//     PlcTask Inputs/GVL_iXlinker.EtherCAT_Master_EPPxxxx.Beckhoff_EPP2xxx.Beckhoff_EPP2xxxEK1122.A_0016_EPP2304_0061_0018.Channel_2.Input <-> Channel 2/Input
//     PlcTask Outputs/GVL_iXlinker.EtherCAT_Master_EPPxxxx.Beckhoff_EPP2xxx.Beckhoff_EPP2xxxEK1122.A_0016_EPP2304_0061_0018.Channel_3.Output <-> Channel 3/Output
//     PlcTask Outputs/GVL_iXlinker.EtherCAT_Master_EPPxxxx.Beckhoff_EPP2xxx.Beckhoff_EPP2xxxEK1122.A_0016_EPP2304_0061_0018.Channel_4.Output <-> Channel 4/Output
//     PlcTask Inputs/GVL_iXlinker.EtherCAT_Master_EPPxxxx.Beckhoff_EPP2xxx.Beckhoff_EPP2xxxEK1122.A_0016_EPP2304_0061_0018.WcState.WcState <-> WcState/WcState
//     PlcTask Inputs/GVL_iXlinker.EtherCAT_Master_EPPxxxx.Beckhoff_EPP2xxx.Beckhoff_EPP2xxxEK1122.A_0016_EPP2304_0061_0018.WcState.InputToggle <-> WcState/InputToggle
//     PlcTask Inputs/GVL_iXlinker.EtherCAT_Master_EPPxxxx.Beckhoff_EPP2xxx.Beckhoff_EPP2xxxEK1122.A_0016_EPP2304_0061_0018.InfoData.State <-> InfoData/State
//   PLC/PLC Instance <-> EtherCAT Master EPPxxxx/Beckhoff EPP2xxx/Beckhoff EPP2xxxEK1122/A_0017(EPP2308-0001-0016)
//     PlcTask Inputs/GVL_iXlinker.EtherCAT_Master_EPPxxxx.Beckhoff_EPP2xxx.Beckhoff_EPP2xxxEK1122.A_0017_EPP2308_0001_0016.Channel_1.Input <-> Channel 1/Input
//     PlcTask Inputs/GVL_iXlinker.EtherCAT_Master_EPPxxxx.Beckhoff_EPP2xxx.Beckhoff_EPP2xxxEK1122.A_0017_EPP2308_0001_0016.Channel_2.Input <-> Channel 2/Input
//     PlcTask Inputs/GVL_iXlinker.EtherCAT_Master_EPPxxxx.Beckhoff_EPP2xxx.Beckhoff_EPP2xxxEK1122.A_0017_EPP2308_0001_0016.Channel_3.Input <-> Channel 3/Input
//     PlcTask Inputs/GVL_iXlinker.EtherCAT_Master_EPPxxxx.Beckhoff_EPP2xxx.Beckhoff_EPP2xxxEK1122.A_0017_EPP2308_0001_0016.Channel_4.Input <-> Channel 4/Input
//     PlcTask Outputs/GVL_iXlinker.EtherCAT_Master_EPPxxxx.Beckhoff_EPP2xxx.Beckhoff_EPP2xxxEK1122.A_0017_EPP2308_0001_0016.Channel_5.Output <-> Channel 5/Output
//     PlcTask Outputs/GVL_iXlinker.EtherCAT_Master_EPPxxxx.Beckhoff_EPP2xxx.Beckhoff_EPP2xxxEK1122.A_0017_EPP2308_0001_0016.Channel_6.Output <-> Channel 6/Output
//     PlcTask Outputs/GVL_iXlinker.EtherCAT_Master_EPPxxxx.Beckhoff_EPP2xxx.Beckhoff_EPP2xxxEK1122.A_0017_EPP2308_0001_0016.Channel_7.Output <-> Channel 7/Output
//     PlcTask Outputs/GVL_iXlinker.EtherCAT_Master_EPPxxxx.Beckhoff_EPP2xxx.Beckhoff_EPP2xxxEK1122.A_0017_EPP2308_0001_0016.Channel_8.Output <-> Channel 8/Output
//     PlcTask Inputs/GVL_iXlinker.EtherCAT_Master_EPPxxxx.Beckhoff_EPP2xxx.Beckhoff_EPP2xxxEK1122.A_0017_EPP2308_0001_0016.WcState.WcState <-> WcState/WcState
//     PlcTask Inputs/GVL_iXlinker.EtherCAT_Master_EPPxxxx.Beckhoff_EPP2xxx.Beckhoff_EPP2xxxEK1122.A_0017_EPP2308_0001_0016.WcState.InputToggle <-> WcState/InputToggle
//     PlcTask Inputs/GVL_iXlinker.EtherCAT_Master_EPPxxxx.Beckhoff_EPP2xxx.Beckhoff_EPP2xxxEK1122.A_0017_EPP2308_0001_0016.InfoData.State <-> InfoData/State
//   PLC/PLC Instance <-> EtherCAT Master EPPxxxx/Beckhoff EPP2xxx/Beckhoff EPP2xxxEK1122/A_0018(EPP2308-0001-0017)
//     PlcTask Inputs/GVL_iXlinker.EtherCAT_Master_EPPxxxx.Beckhoff_EPP2xxx.Beckhoff_EPP2xxxEK1122.A_0018_EPP2308_0001_0017.Channel_1.Input <-> Channel 1/Input
//     PlcTask Inputs/GVL_iXlinker.EtherCAT_Master_EPPxxxx.Beckhoff_EPP2xxx.Beckhoff_EPP2xxxEK1122.A_0018_EPP2308_0001_0017.Channel_2.Input <-> Channel 2/Input
//     PlcTask Inputs/GVL_iXlinker.EtherCAT_Master_EPPxxxx.Beckhoff_EPP2xxx.Beckhoff_EPP2xxxEK1122.A_0018_EPP2308_0001_0017.Channel_3.Input <-> Channel 3/Input
//     PlcTask Inputs/GVL_iXlinker.EtherCAT_Master_EPPxxxx.Beckhoff_EPP2xxx.Beckhoff_EPP2xxxEK1122.A_0018_EPP2308_0001_0017.Channel_4.Input <-> Channel 4/Input
//     PlcTask Outputs/GVL_iXlinker.EtherCAT_Master_EPPxxxx.Beckhoff_EPP2xxx.Beckhoff_EPP2xxxEK1122.A_0018_EPP2308_0001_0017.Channel_5.Output <-> Channel 5/Output
//     PlcTask Outputs/GVL_iXlinker.EtherCAT_Master_EPPxxxx.Beckhoff_EPP2xxx.Beckhoff_EPP2xxxEK1122.A_0018_EPP2308_0001_0017.Channel_6.Output <-> Channel 6/Output
//     PlcTask Outputs/GVL_iXlinker.EtherCAT_Master_EPPxxxx.Beckhoff_EPP2xxx.Beckhoff_EPP2xxxEK1122.A_0018_EPP2308_0001_0017.Channel_7.Output <-> Channel 7/Output
//     PlcTask Outputs/GVL_iXlinker.EtherCAT_Master_EPPxxxx.Beckhoff_EPP2xxx.Beckhoff_EPP2xxxEK1122.A_0018_EPP2308_0001_0017.Channel_8.Output <-> Channel 8/Output
//     PlcTask Inputs/GVL_iXlinker.EtherCAT_Master_EPPxxxx.Beckhoff_EPP2xxx.Beckhoff_EPP2xxxEK1122.A_0018_EPP2308_0001_0017.WcState.WcState <-> WcState/WcState
//     PlcTask Inputs/GVL_iXlinker.EtherCAT_Master_EPPxxxx.Beckhoff_EPP2xxx.Beckhoff_EPP2xxxEK1122.A_0018_EPP2308_0001_0017.WcState.InputToggle <-> WcState/InputToggle
//     PlcTask Inputs/GVL_iXlinker.EtherCAT_Master_EPPxxxx.Beckhoff_EPP2xxx.Beckhoff_EPP2xxxEK1122.A_0018_EPP2308_0001_0017.InfoData.State <-> InfoData/State
//   PLC/PLC Instance <-> EtherCAT Master EPPxxxx/Beckhoff EPP2xxx/Beckhoff EPP2xxxEK1122/A_0019(EPP2308-0001-0018)
//     PlcTask Inputs/GVL_iXlinker.EtherCAT_Master_EPPxxxx.Beckhoff_EPP2xxx.Beckhoff_EPP2xxxEK1122.A_0019_EPP2308_0001_0018.Channel_1.Input <-> Channel 1/Input
//     PlcTask Inputs/GVL_iXlinker.EtherCAT_Master_EPPxxxx.Beckhoff_EPP2xxx.Beckhoff_EPP2xxxEK1122.A_0019_EPP2308_0001_0018.Channel_2.Input <-> Channel 2/Input
//     PlcTask Inputs/GVL_iXlinker.EtherCAT_Master_EPPxxxx.Beckhoff_EPP2xxx.Beckhoff_EPP2xxxEK1122.A_0019_EPP2308_0001_0018.Channel_3.Input <-> Channel 3/Input
//     PlcTask Inputs/GVL_iXlinker.EtherCAT_Master_EPPxxxx.Beckhoff_EPP2xxx.Beckhoff_EPP2xxxEK1122.A_0019_EPP2308_0001_0018.Channel_4.Input <-> Channel 4/Input
//     PlcTask Outputs/GVL_iXlinker.EtherCAT_Master_EPPxxxx.Beckhoff_EPP2xxx.Beckhoff_EPP2xxxEK1122.A_0019_EPP2308_0001_0018.Channel_5.Output <-> Channel 5/Output
//     PlcTask Outputs/GVL_iXlinker.EtherCAT_Master_EPPxxxx.Beckhoff_EPP2xxx.Beckhoff_EPP2xxxEK1122.A_0019_EPP2308_0001_0018.Channel_6.Output <-> Channel 6/Output
//     PlcTask Outputs/GVL_iXlinker.EtherCAT_Master_EPPxxxx.Beckhoff_EPP2xxx.Beckhoff_EPP2xxxEK1122.A_0019_EPP2308_0001_0018.Channel_7.Output <-> Channel 7/Output
//     PlcTask Outputs/GVL_iXlinker.EtherCAT_Master_EPPxxxx.Beckhoff_EPP2xxx.Beckhoff_EPP2xxxEK1122.A_0019_EPP2308_0001_0018.Channel_8.Output <-> Channel 8/Output
//     PlcTask Inputs/GVL_iXlinker.EtherCAT_Master_EPPxxxx.Beckhoff_EPP2xxx.Beckhoff_EPP2xxxEK1122.A_0019_EPP2308_0001_0018.WcState.WcState <-> WcState/WcState
//     PlcTask Inputs/GVL_iXlinker.EtherCAT_Master_EPPxxxx.Beckhoff_EPP2xxx.Beckhoff_EPP2xxxEK1122.A_0019_EPP2308_0001_0018.WcState.InputToggle <-> WcState/InputToggle
//     PlcTask Inputs/GVL_iXlinker.EtherCAT_Master_EPPxxxx.Beckhoff_EPP2xxx.Beckhoff_EPP2xxxEK1122.A_0019_EPP2308_0001_0018.InfoData.State <-> InfoData/State
//   PLC/PLC Instance <-> EtherCAT Master EPPxxxx/Beckhoff EPP2xxx/Beckhoff EPP2xxxEK1122/A_0020(EPP2308-0002-0016)
//     PlcTask Inputs/GVL_iXlinker.EtherCAT_Master_EPPxxxx.Beckhoff_EPP2xxx.Beckhoff_EPP2xxxEK1122.A_0020_EPP2308_0002_0016.Channel_1.Input <-> Channel 1/Input
//     PlcTask Inputs/GVL_iXlinker.EtherCAT_Master_EPPxxxx.Beckhoff_EPP2xxx.Beckhoff_EPP2xxxEK1122.A_0020_EPP2308_0002_0016.Channel_2.Input <-> Channel 2/Input
//     PlcTask Inputs/GVL_iXlinker.EtherCAT_Master_EPPxxxx.Beckhoff_EPP2xxx.Beckhoff_EPP2xxxEK1122.A_0020_EPP2308_0002_0016.Channel_3.Input <-> Channel 3/Input
//     PlcTask Inputs/GVL_iXlinker.EtherCAT_Master_EPPxxxx.Beckhoff_EPP2xxx.Beckhoff_EPP2xxxEK1122.A_0020_EPP2308_0002_0016.Channel_4.Input <-> Channel 4/Input
//     PlcTask Outputs/GVL_iXlinker.EtherCAT_Master_EPPxxxx.Beckhoff_EPP2xxx.Beckhoff_EPP2xxxEK1122.A_0020_EPP2308_0002_0016.Channel_5.Output <-> Channel 5/Output
//     PlcTask Outputs/GVL_iXlinker.EtherCAT_Master_EPPxxxx.Beckhoff_EPP2xxx.Beckhoff_EPP2xxxEK1122.A_0020_EPP2308_0002_0016.Channel_6.Output <-> Channel 6/Output
//     PlcTask Outputs/GVL_iXlinker.EtherCAT_Master_EPPxxxx.Beckhoff_EPP2xxx.Beckhoff_EPP2xxxEK1122.A_0020_EPP2308_0002_0016.Channel_7.Output <-> Channel 7/Output
//     PlcTask Outputs/GVL_iXlinker.EtherCAT_Master_EPPxxxx.Beckhoff_EPP2xxx.Beckhoff_EPP2xxxEK1122.A_0020_EPP2308_0002_0016.Channel_8.Output <-> Channel 8/Output
//     PlcTask Inputs/GVL_iXlinker.EtherCAT_Master_EPPxxxx.Beckhoff_EPP2xxx.Beckhoff_EPP2xxxEK1122.A_0020_EPP2308_0002_0016.WcState.WcState <-> WcState/WcState
//     PlcTask Inputs/GVL_iXlinker.EtherCAT_Master_EPPxxxx.Beckhoff_EPP2xxx.Beckhoff_EPP2xxxEK1122.A_0020_EPP2308_0002_0016.WcState.InputToggle <-> WcState/InputToggle
//     PlcTask Inputs/GVL_iXlinker.EtherCAT_Master_EPPxxxx.Beckhoff_EPP2xxx.Beckhoff_EPP2xxxEK1122.A_0020_EPP2308_0002_0016.InfoData.State <-> InfoData/State
//   PLC/PLC Instance <-> EtherCAT Master EPPxxxx/Beckhoff EPP2xxx/Beckhoff EPP2xxxEK1122/A_0021(EPP2308-0002-0017)
//     PlcTask Inputs/GVL_iXlinker.EtherCAT_Master_EPPxxxx.Beckhoff_EPP2xxx.Beckhoff_EPP2xxxEK1122.A_0021_EPP2308_0002_0017.Channel_1.Input <-> Channel 1/Input
//     PlcTask Inputs/GVL_iXlinker.EtherCAT_Master_EPPxxxx.Beckhoff_EPP2xxx.Beckhoff_EPP2xxxEK1122.A_0021_EPP2308_0002_0017.Channel_2.Input <-> Channel 2/Input
//     PlcTask Inputs/GVL_iXlinker.EtherCAT_Master_EPPxxxx.Beckhoff_EPP2xxx.Beckhoff_EPP2xxxEK1122.A_0021_EPP2308_0002_0017.Channel_3.Input <-> Channel 3/Input
//     PlcTask Inputs/GVL_iXlinker.EtherCAT_Master_EPPxxxx.Beckhoff_EPP2xxx.Beckhoff_EPP2xxxEK1122.A_0021_EPP2308_0002_0017.Channel_4.Input <-> Channel 4/Input
//     PlcTask Outputs/GVL_iXlinker.EtherCAT_Master_EPPxxxx.Beckhoff_EPP2xxx.Beckhoff_EPP2xxxEK1122.A_0021_EPP2308_0002_0017.Channel_5.Output <-> Channel 5/Output
//     PlcTask Outputs/GVL_iXlinker.EtherCAT_Master_EPPxxxx.Beckhoff_EPP2xxx.Beckhoff_EPP2xxxEK1122.A_0021_EPP2308_0002_0017.Channel_6.Output <-> Channel 6/Output
//     PlcTask Outputs/GVL_iXlinker.EtherCAT_Master_EPPxxxx.Beckhoff_EPP2xxx.Beckhoff_EPP2xxxEK1122.A_0021_EPP2308_0002_0017.Channel_7.Output <-> Channel 7/Output
//     PlcTask Outputs/GVL_iXlinker.EtherCAT_Master_EPPxxxx.Beckhoff_EPP2xxx.Beckhoff_EPP2xxxEK1122.A_0021_EPP2308_0002_0017.Channel_8.Output <-> Channel 8/Output
//     PlcTask Inputs/GVL_iXlinker.EtherCAT_Master_EPPxxxx.Beckhoff_EPP2xxx.Beckhoff_EPP2xxxEK1122.A_0021_EPP2308_0002_0017.WcState.WcState <-> WcState/WcState
//     PlcTask Inputs/GVL_iXlinker.EtherCAT_Master_EPPxxxx.Beckhoff_EPP2xxx.Beckhoff_EPP2xxxEK1122.A_0021_EPP2308_0002_0017.WcState.InputToggle <-> WcState/InputToggle
//     PlcTask Inputs/GVL_iXlinker.EtherCAT_Master_EPPxxxx.Beckhoff_EPP2xxx.Beckhoff_EPP2xxxEK1122.A_0021_EPP2308_0002_0017.InfoData.State <-> InfoData/State
//   PLC/PLC Instance <-> EtherCAT Master EPPxxxx/Beckhoff EPP2xxx/Beckhoff EPP2xxxEK1122/A_0022(EPP2308-0002-0018)
//     PlcTask Inputs/GVL_iXlinker.EtherCAT_Master_EPPxxxx.Beckhoff_EPP2xxx.Beckhoff_EPP2xxxEK1122.A_0022_EPP2308_0002_0018.Channel_1.Input <-> Channel 1/Input
//     PlcTask Inputs/GVL_iXlinker.EtherCAT_Master_EPPxxxx.Beckhoff_EPP2xxx.Beckhoff_EPP2xxxEK1122.A_0022_EPP2308_0002_0018.Channel_2.Input <-> Channel 2/Input
//     PlcTask Inputs/GVL_iXlinker.EtherCAT_Master_EPPxxxx.Beckhoff_EPP2xxx.Beckhoff_EPP2xxxEK1122.A_0022_EPP2308_0002_0018.Channel_3.Input <-> Channel 3/Input
//     PlcTask Inputs/GVL_iXlinker.EtherCAT_Master_EPPxxxx.Beckhoff_EPP2xxx.Beckhoff_EPP2xxxEK1122.A_0022_EPP2308_0002_0018.Channel_4.Input <-> Channel 4/Input
//     PlcTask Outputs/GVL_iXlinker.EtherCAT_Master_EPPxxxx.Beckhoff_EPP2xxx.Beckhoff_EPP2xxxEK1122.A_0022_EPP2308_0002_0018.Channel_5.Output <-> Channel 5/Output
//     PlcTask Outputs/GVL_iXlinker.EtherCAT_Master_EPPxxxx.Beckhoff_EPP2xxx.Beckhoff_EPP2xxxEK1122.A_0022_EPP2308_0002_0018.Channel_6.Output <-> Channel 6/Output
//     PlcTask Outputs/GVL_iXlinker.EtherCAT_Master_EPPxxxx.Beckhoff_EPP2xxx.Beckhoff_EPP2xxxEK1122.A_0022_EPP2308_0002_0018.Channel_7.Output <-> Channel 7/Output
//     PlcTask Outputs/GVL_iXlinker.EtherCAT_Master_EPPxxxx.Beckhoff_EPP2xxx.Beckhoff_EPP2xxxEK1122.A_0022_EPP2308_0002_0018.Channel_8.Output <-> Channel 8/Output
//     PlcTask Inputs/GVL_iXlinker.EtherCAT_Master_EPPxxxx.Beckhoff_EPP2xxx.Beckhoff_EPP2xxxEK1122.A_0022_EPP2308_0002_0018.WcState.WcState <-> WcState/WcState
//     PlcTask Inputs/GVL_iXlinker.EtherCAT_Master_EPPxxxx.Beckhoff_EPP2xxx.Beckhoff_EPP2xxxEK1122.A_0022_EPP2308_0002_0018.WcState.InputToggle <-> WcState/InputToggle
//     PlcTask Inputs/GVL_iXlinker.EtherCAT_Master_EPPxxxx.Beckhoff_EPP2xxx.Beckhoff_EPP2xxxEK1122.A_0022_EPP2308_0002_0018.InfoData.State <-> InfoData/State
//   PLC/PLC Instance <-> EtherCAT Master EPPxxxx/Beckhoff EPP2xxx/Beckhoff EPP2xxxEK1122/A_0023(EPP2316-0003-0016)
//     PlcTask Inputs/GVL_iXlinker.EtherCAT_Master_EPPxxxx.Beckhoff_EPP2xxx.Beckhoff_EPP2xxxEK1122.A_0023_EPP2316_0003_0016.DIG_Inputs.Input[0] <-> DIG Inputs/Input 1
//     PlcTask Inputs/GVL_iXlinker.EtherCAT_Master_EPPxxxx.Beckhoff_EPP2xxx.Beckhoff_EPP2xxxEK1122.A_0023_EPP2316_0003_0016.DIG_Inputs.Input[1] <-> DIG Inputs/Input 2
//     PlcTask Inputs/GVL_iXlinker.EtherCAT_Master_EPPxxxx.Beckhoff_EPP2xxx.Beckhoff_EPP2xxxEK1122.A_0023_EPP2316_0003_0016.DIG_Inputs.Input[2] <-> DIG Inputs/Input 3
//     PlcTask Inputs/GVL_iXlinker.EtherCAT_Master_EPPxxxx.Beckhoff_EPP2xxx.Beckhoff_EPP2xxxEK1122.A_0023_EPP2316_0003_0016.DIG_Inputs.Input[3] <-> DIG Inputs/Input 4
//     PlcTask Inputs/GVL_iXlinker.EtherCAT_Master_EPPxxxx.Beckhoff_EPP2xxx.Beckhoff_EPP2xxxEK1122.A_0023_EPP2316_0003_0016.DIG_Inputs.Input[4] <-> DIG Inputs/Input 5
//     PlcTask Inputs/GVL_iXlinker.EtherCAT_Master_EPPxxxx.Beckhoff_EPP2xxx.Beckhoff_EPP2xxxEK1122.A_0023_EPP2316_0003_0016.DIG_Inputs.Input[5] <-> DIG Inputs/Input 6
//     PlcTask Inputs/GVL_iXlinker.EtherCAT_Master_EPPxxxx.Beckhoff_EPP2xxx.Beckhoff_EPP2xxxEK1122.A_0023_EPP2316_0003_0016.DIG_Inputs.Input[6] <-> DIG Inputs/Input 7
//     PlcTask Inputs/GVL_iXlinker.EtherCAT_Master_EPPxxxx.Beckhoff_EPP2xxx.Beckhoff_EPP2xxxEK1122.A_0023_EPP2316_0003_0016.DIG_Inputs.Input[7] <-> DIG Inputs/Input 8
//     PlcTask Inputs/GVL_iXlinker.EtherCAT_Master_EPPxxxx.Beckhoff_EPP2xxx.Beckhoff_EPP2xxxEK1122.A_0023_EPP2316_0003_0016.DIG_Inputs.Sync_Error <-> DIG Inputs/Sync Error
//     PlcTask Inputs/GVL_iXlinker.EtherCAT_Master_EPPxxxx.Beckhoff_EPP2xxx.Beckhoff_EPP2xxxEK1122.A_0023_EPP2316_0003_0016.DIG_Diag_Inputs.Diag_Input[0] <-> DIG Diag Inputs/Diag Input 1
//     PlcTask Inputs/GVL_iXlinker.EtherCAT_Master_EPPxxxx.Beckhoff_EPP2xxx.Beckhoff_EPP2xxxEK1122.A_0023_EPP2316_0003_0016.DIG_Diag_Inputs.Diag_Input[1] <-> DIG Diag Inputs/Diag Input 2
//     PlcTask Inputs/GVL_iXlinker.EtherCAT_Master_EPPxxxx.Beckhoff_EPP2xxx.Beckhoff_EPP2xxxEK1122.A_0023_EPP2316_0003_0016.DIG_Diag_Inputs.Diag_Input[2] <-> DIG Diag Inputs/Diag Input 3
//     PlcTask Inputs/GVL_iXlinker.EtherCAT_Master_EPPxxxx.Beckhoff_EPP2xxx.Beckhoff_EPP2xxxEK1122.A_0023_EPP2316_0003_0016.DIG_Diag_Inputs.Diag_Input[3] <-> DIG Diag Inputs/Diag Input 4
//     PlcTask Inputs/GVL_iXlinker.EtherCAT_Master_EPPxxxx.Beckhoff_EPP2xxx.Beckhoff_EPP2xxxEK1122.A_0023_EPP2316_0003_0016.DIG_Diag_Inputs.Diag_Input[4] <-> DIG Diag Inputs/Diag Input 5
//     PlcTask Inputs/GVL_iXlinker.EtherCAT_Master_EPPxxxx.Beckhoff_EPP2xxx.Beckhoff_EPP2xxxEK1122.A_0023_EPP2316_0003_0016.DIG_Diag_Inputs.Diag_Input[5] <-> DIG Diag Inputs/Diag Input 6
//     PlcTask Inputs/GVL_iXlinker.EtherCAT_Master_EPPxxxx.Beckhoff_EPP2xxx.Beckhoff_EPP2xxxEK1122.A_0023_EPP2316_0003_0016.DIG_Diag_Inputs.Diag_Input[6] <-> DIG Diag Inputs/Diag Input 7
//     PlcTask Inputs/GVL_iXlinker.EtherCAT_Master_EPPxxxx.Beckhoff_EPP2xxx.Beckhoff_EPP2xxxEK1122.A_0023_EPP2316_0003_0016.DIG_Diag_Inputs.Diag_Input[7] <-> DIG Diag Inputs/Diag Input 8
//     PlcTask Inputs/GVL_iXlinker.EtherCAT_Master_EPPxxxx.Beckhoff_EPP2xxx.Beckhoff_EPP2xxxEK1122.A_0023_EPP2316_0003_0016.DIG_Inputs_Device.Safe_state_active <-> DIG Inputs Device/Safe state active
//     PlcTask Inputs/GVL_iXlinker.EtherCAT_Master_EPPxxxx.Beckhoff_EPP2xxx.Beckhoff_EPP2xxxEK1122.A_0023_EPP2316_0003_0016.DIG_Inputs_Device.Error_channel[0] <-> DIG Inputs Device/Error channel 1
//     PlcTask Inputs/GVL_iXlinker.EtherCAT_Master_EPPxxxx.Beckhoff_EPP2xxx.Beckhoff_EPP2xxxEK1122.A_0023_EPP2316_0003_0016.DIG_Inputs_Device.Error_channel[1] <-> DIG Inputs Device/Error channel 2
//     PlcTask Inputs/GVL_iXlinker.EtherCAT_Master_EPPxxxx.Beckhoff_EPP2xxx.Beckhoff_EPP2xxxEK1122.A_0023_EPP2316_0003_0016.DIG_Inputs_Device.Sync_error <-> DIG Inputs Device/Sync error
//     PlcTask Inputs/GVL_iXlinker.EtherCAT_Master_EPPxxxx.Beckhoff_EPP2xxx.Beckhoff_EPP2xxxEK1122.A_0023_EPP2316_0003_0016.DIG_Inputs_Device.TxPDO_Toggle <-> DIG Inputs Device/TxPDO Toggle
//     PlcTask Outputs/GVL_iXlinker.EtherCAT_Master_EPPxxxx.Beckhoff_EPP2xxx.Beckhoff_EPP2xxxEK1122.A_0023_EPP2316_0003_0016.DIG_Outputs.Output[0] <-> DIG Outputs/Output 1
//     PlcTask Outputs/GVL_iXlinker.EtherCAT_Master_EPPxxxx.Beckhoff_EPP2xxx.Beckhoff_EPP2xxxEK1122.A_0023_EPP2316_0003_0016.DIG_Outputs.Output[1] <-> DIG Outputs/Output 2
//     PlcTask Outputs/GVL_iXlinker.EtherCAT_Master_EPPxxxx.Beckhoff_EPP2xxx.Beckhoff_EPP2xxxEK1122.A_0023_EPP2316_0003_0016.DIG_Outputs.Output[2] <-> DIG Outputs/Output 3
//     PlcTask Outputs/GVL_iXlinker.EtherCAT_Master_EPPxxxx.Beckhoff_EPP2xxx.Beckhoff_EPP2xxxEK1122.A_0023_EPP2316_0003_0016.DIG_Outputs.Output[3] <-> DIG Outputs/Output 4
//     PlcTask Outputs/GVL_iXlinker.EtherCAT_Master_EPPxxxx.Beckhoff_EPP2xxx.Beckhoff_EPP2xxxEK1122.A_0023_EPP2316_0003_0016.DIG_Outputs.Output[4] <-> DIG Outputs/Output 5
//     PlcTask Outputs/GVL_iXlinker.EtherCAT_Master_EPPxxxx.Beckhoff_EPP2xxx.Beckhoff_EPP2xxxEK1122.A_0023_EPP2316_0003_0016.DIG_Outputs.Output[5] <-> DIG Outputs/Output 6
//     PlcTask Outputs/GVL_iXlinker.EtherCAT_Master_EPPxxxx.Beckhoff_EPP2xxx.Beckhoff_EPP2xxxEK1122.A_0023_EPP2316_0003_0016.DIG_Outputs.Output[6] <-> DIG Outputs/Output 7
//     PlcTask Outputs/GVL_iXlinker.EtherCAT_Master_EPPxxxx.Beckhoff_EPP2xxx.Beckhoff_EPP2xxxEK1122.A_0023_EPP2316_0003_0016.DIG_Outputs.Output[7] <-> DIG Outputs/Output 8
//     PlcTask Outputs/GVL_iXlinker.EtherCAT_Master_EPPxxxx.Beckhoff_EPP2xxx.Beckhoff_EPP2xxxEK1122.A_0023_EPP2316_0003_0016.DIG_Outputs_Device.Set_safe_state <-> DIG Outputs Device/Set safe state
//     PlcTask Outputs/GVL_iXlinker.EtherCAT_Master_EPPxxxx.Beckhoff_EPP2xxx.Beckhoff_EPP2xxxEK1122.A_0023_EPP2316_0003_0016.DIG_Outputs_Device.Reset_outputs <-> DIG Outputs Device/Reset outputs
//     PlcTask Inputs/GVL_iXlinker.EtherCAT_Master_EPPxxxx.Beckhoff_EPP2xxx.Beckhoff_EPP2xxxEK1122.A_0023_EPP2316_0003_0016.WcState.WcState <-> WcState/WcState
//     PlcTask Inputs/GVL_iXlinker.EtherCAT_Master_EPPxxxx.Beckhoff_EPP2xxx.Beckhoff_EPP2xxxEK1122.A_0023_EPP2316_0003_0016.WcState.InputToggle <-> WcState/InputToggle
//     PlcTask Inputs/GVL_iXlinker.EtherCAT_Master_EPPxxxx.Beckhoff_EPP2xxx.Beckhoff_EPP2xxxEK1122.A_0023_EPP2316_0003_0016.InfoData.AdsAddr <-> InfoData/AdsAddr
//     PlcTask Inputs/GVL_iXlinker.EtherCAT_Master_EPPxxxx.Beckhoff_EPP2xxx.Beckhoff_EPP2xxxEK1122.A_0023_EPP2316_0003_0016.InfoData.State <-> InfoData/State
//   PLC/PLC Instance <-> EtherCAT Master EPPxxxx/Beckhoff EPP2xxx/Beckhoff EPP2xxxEK1122/A_0024(EPP2316-0003-0017)
//     PlcTask Inputs/GVL_iXlinker.EtherCAT_Master_EPPxxxx.Beckhoff_EPP2xxx.Beckhoff_EPP2xxxEK1122.A_0024_EPP2316_0003_0017.DIG_Inputs.Input[0] <-> DIG Inputs/Input 1
//     PlcTask Inputs/GVL_iXlinker.EtherCAT_Master_EPPxxxx.Beckhoff_EPP2xxx.Beckhoff_EPP2xxxEK1122.A_0024_EPP2316_0003_0017.DIG_Inputs.Input[1] <-> DIG Inputs/Input 2
//     PlcTask Inputs/GVL_iXlinker.EtherCAT_Master_EPPxxxx.Beckhoff_EPP2xxx.Beckhoff_EPP2xxxEK1122.A_0024_EPP2316_0003_0017.DIG_Inputs.Input[2] <-> DIG Inputs/Input 3
//     PlcTask Inputs/GVL_iXlinker.EtherCAT_Master_EPPxxxx.Beckhoff_EPP2xxx.Beckhoff_EPP2xxxEK1122.A_0024_EPP2316_0003_0017.DIG_Inputs.Input[3] <-> DIG Inputs/Input 4
//     PlcTask Inputs/GVL_iXlinker.EtherCAT_Master_EPPxxxx.Beckhoff_EPP2xxx.Beckhoff_EPP2xxxEK1122.A_0024_EPP2316_0003_0017.DIG_Inputs.Input[4] <-> DIG Inputs/Input 5
//     PlcTask Inputs/GVL_iXlinker.EtherCAT_Master_EPPxxxx.Beckhoff_EPP2xxx.Beckhoff_EPP2xxxEK1122.A_0024_EPP2316_0003_0017.DIG_Inputs.Input[5] <-> DIG Inputs/Input 6
//     PlcTask Inputs/GVL_iXlinker.EtherCAT_Master_EPPxxxx.Beckhoff_EPP2xxx.Beckhoff_EPP2xxxEK1122.A_0024_EPP2316_0003_0017.DIG_Inputs.Input[6] <-> DIG Inputs/Input 7
//     PlcTask Inputs/GVL_iXlinker.EtherCAT_Master_EPPxxxx.Beckhoff_EPP2xxx.Beckhoff_EPP2xxxEK1122.A_0024_EPP2316_0003_0017.DIG_Inputs.Input[7] <-> DIG Inputs/Input 8
//     PlcTask Inputs/GVL_iXlinker.EtherCAT_Master_EPPxxxx.Beckhoff_EPP2xxx.Beckhoff_EPP2xxxEK1122.A_0024_EPP2316_0003_0017.DIG_Inputs.Sync_Error <-> DIG Inputs/Sync Error
//     PlcTask Inputs/GVL_iXlinker.EtherCAT_Master_EPPxxxx.Beckhoff_EPP2xxx.Beckhoff_EPP2xxxEK1122.A_0024_EPP2316_0003_0017.DIG_Diag_Inputs.Diag_Input[0] <-> DIG Diag Inputs/Diag Input 1
//     PlcTask Inputs/GVL_iXlinker.EtherCAT_Master_EPPxxxx.Beckhoff_EPP2xxx.Beckhoff_EPP2xxxEK1122.A_0024_EPP2316_0003_0017.DIG_Diag_Inputs.Diag_Input[1] <-> DIG Diag Inputs/Diag Input 2
//     PlcTask Inputs/GVL_iXlinker.EtherCAT_Master_EPPxxxx.Beckhoff_EPP2xxx.Beckhoff_EPP2xxxEK1122.A_0024_EPP2316_0003_0017.DIG_Diag_Inputs.Diag_Input[2] <-> DIG Diag Inputs/Diag Input 3
//     PlcTask Inputs/GVL_iXlinker.EtherCAT_Master_EPPxxxx.Beckhoff_EPP2xxx.Beckhoff_EPP2xxxEK1122.A_0024_EPP2316_0003_0017.DIG_Diag_Inputs.Diag_Input[3] <-> DIG Diag Inputs/Diag Input 4
//     PlcTask Inputs/GVL_iXlinker.EtherCAT_Master_EPPxxxx.Beckhoff_EPP2xxx.Beckhoff_EPP2xxxEK1122.A_0024_EPP2316_0003_0017.DIG_Diag_Inputs.Diag_Input[4] <-> DIG Diag Inputs/Diag Input 5
//     PlcTask Inputs/GVL_iXlinker.EtherCAT_Master_EPPxxxx.Beckhoff_EPP2xxx.Beckhoff_EPP2xxxEK1122.A_0024_EPP2316_0003_0017.DIG_Diag_Inputs.Diag_Input[5] <-> DIG Diag Inputs/Diag Input 6
//     PlcTask Inputs/GVL_iXlinker.EtherCAT_Master_EPPxxxx.Beckhoff_EPP2xxx.Beckhoff_EPP2xxxEK1122.A_0024_EPP2316_0003_0017.DIG_Diag_Inputs.Diag_Input[6] <-> DIG Diag Inputs/Diag Input 7
//     PlcTask Inputs/GVL_iXlinker.EtherCAT_Master_EPPxxxx.Beckhoff_EPP2xxx.Beckhoff_EPP2xxxEK1122.A_0024_EPP2316_0003_0017.DIG_Diag_Inputs.Diag_Input[7] <-> DIG Diag Inputs/Diag Input 8
//     PlcTask Inputs/GVL_iXlinker.EtherCAT_Master_EPPxxxx.Beckhoff_EPP2xxx.Beckhoff_EPP2xxxEK1122.A_0024_EPP2316_0003_0017.DIG_Inputs_Device.Safe_state_active <-> DIG Inputs Device/Safe state active
//     PlcTask Inputs/GVL_iXlinker.EtherCAT_Master_EPPxxxx.Beckhoff_EPP2xxx.Beckhoff_EPP2xxxEK1122.A_0024_EPP2316_0003_0017.DIG_Inputs_Device.Error_channel[0] <-> DIG Inputs Device/Error channel 1
//     PlcTask Inputs/GVL_iXlinker.EtherCAT_Master_EPPxxxx.Beckhoff_EPP2xxx.Beckhoff_EPP2xxxEK1122.A_0024_EPP2316_0003_0017.DIG_Inputs_Device.Error_channel[1] <-> DIG Inputs Device/Error channel 2
//     PlcTask Inputs/GVL_iXlinker.EtherCAT_Master_EPPxxxx.Beckhoff_EPP2xxx.Beckhoff_EPP2xxxEK1122.A_0024_EPP2316_0003_0017.DIG_Inputs_Device.Sync_error <-> DIG Inputs Device/Sync error
//     PlcTask Inputs/GVL_iXlinker.EtherCAT_Master_EPPxxxx.Beckhoff_EPP2xxx.Beckhoff_EPP2xxxEK1122.A_0024_EPP2316_0003_0017.DIG_Inputs_Device.TxPDO_Toggle <-> DIG Inputs Device/TxPDO Toggle
//     PlcTask Outputs/GVL_iXlinker.EtherCAT_Master_EPPxxxx.Beckhoff_EPP2xxx.Beckhoff_EPP2xxxEK1122.A_0024_EPP2316_0003_0017.DIG_Outputs.Output[0] <-> DIG Outputs/Output 1
//     PlcTask Outputs/GVL_iXlinker.EtherCAT_Master_EPPxxxx.Beckhoff_EPP2xxx.Beckhoff_EPP2xxxEK1122.A_0024_EPP2316_0003_0017.DIG_Outputs.Output[1] <-> DIG Outputs/Output 2
//     PlcTask Outputs/GVL_iXlinker.EtherCAT_Master_EPPxxxx.Beckhoff_EPP2xxx.Beckhoff_EPP2xxxEK1122.A_0024_EPP2316_0003_0017.DIG_Outputs.Output[2] <-> DIG Outputs/Output 3
//     PlcTask Outputs/GVL_iXlinker.EtherCAT_Master_EPPxxxx.Beckhoff_EPP2xxx.Beckhoff_EPP2xxxEK1122.A_0024_EPP2316_0003_0017.DIG_Outputs.Output[3] <-> DIG Outputs/Output 4
//     PlcTask Outputs/GVL_iXlinker.EtherCAT_Master_EPPxxxx.Beckhoff_EPP2xxx.Beckhoff_EPP2xxxEK1122.A_0024_EPP2316_0003_0017.DIG_Outputs.Output[4] <-> DIG Outputs/Output 5
//     PlcTask Outputs/GVL_iXlinker.EtherCAT_Master_EPPxxxx.Beckhoff_EPP2xxx.Beckhoff_EPP2xxxEK1122.A_0024_EPP2316_0003_0017.DIG_Outputs.Output[5] <-> DIG Outputs/Output 6
//     PlcTask Outputs/GVL_iXlinker.EtherCAT_Master_EPPxxxx.Beckhoff_EPP2xxx.Beckhoff_EPP2xxxEK1122.A_0024_EPP2316_0003_0017.DIG_Outputs.Output[6] <-> DIG Outputs/Output 7
//     PlcTask Outputs/GVL_iXlinker.EtherCAT_Master_EPPxxxx.Beckhoff_EPP2xxx.Beckhoff_EPP2xxxEK1122.A_0024_EPP2316_0003_0017.DIG_Outputs.Output[7] <-> DIG Outputs/Output 8
//     PlcTask Outputs/GVL_iXlinker.EtherCAT_Master_EPPxxxx.Beckhoff_EPP2xxx.Beckhoff_EPP2xxxEK1122.A_0024_EPP2316_0003_0017.DIG_Outputs_Device.Set_safe_state <-> DIG Outputs Device/Set safe state
//     PlcTask Outputs/GVL_iXlinker.EtherCAT_Master_EPPxxxx.Beckhoff_EPP2xxx.Beckhoff_EPP2xxxEK1122.A_0024_EPP2316_0003_0017.DIG_Outputs_Device.Reset_outputs <-> DIG Outputs Device/Reset outputs
//     PlcTask Inputs/GVL_iXlinker.EtherCAT_Master_EPPxxxx.Beckhoff_EPP2xxx.Beckhoff_EPP2xxxEK1122.A_0024_EPP2316_0003_0017.WcState.WcState <-> WcState/WcState
//     PlcTask Inputs/GVL_iXlinker.EtherCAT_Master_EPPxxxx.Beckhoff_EPP2xxx.Beckhoff_EPP2xxxEK1122.A_0024_EPP2316_0003_0017.WcState.InputToggle <-> WcState/InputToggle
//     PlcTask Inputs/GVL_iXlinker.EtherCAT_Master_EPPxxxx.Beckhoff_EPP2xxx.Beckhoff_EPP2xxxEK1122.A_0024_EPP2316_0003_0017.InfoData.AdsAddr <-> InfoData/AdsAddr
//     PlcTask Inputs/GVL_iXlinker.EtherCAT_Master_EPPxxxx.Beckhoff_EPP2xxx.Beckhoff_EPP2xxxEK1122.A_0024_EPP2316_0003_0017.InfoData.State <-> InfoData/State
//   PLC/PLC Instance <-> EtherCAT Master EPPxxxx/Beckhoff EPP2xxx/Beckhoff EPP2xxxEK1122/A_0025(EPP2316-0003-0018)
//     PlcTask Inputs/GVL_iXlinker.EtherCAT_Master_EPPxxxx.Beckhoff_EPP2xxx.Beckhoff_EPP2xxxEK1122.A_0025_EPP2316_0003_0018.DIG_Inputs.Input[0] <-> DIG Inputs/Input 1
//     PlcTask Inputs/GVL_iXlinker.EtherCAT_Master_EPPxxxx.Beckhoff_EPP2xxx.Beckhoff_EPP2xxxEK1122.A_0025_EPP2316_0003_0018.DIG_Inputs.Input[1] <-> DIG Inputs/Input 2
//     PlcTask Inputs/GVL_iXlinker.EtherCAT_Master_EPPxxxx.Beckhoff_EPP2xxx.Beckhoff_EPP2xxxEK1122.A_0025_EPP2316_0003_0018.DIG_Inputs.Input[2] <-> DIG Inputs/Input 3
//     PlcTask Inputs/GVL_iXlinker.EtherCAT_Master_EPPxxxx.Beckhoff_EPP2xxx.Beckhoff_EPP2xxxEK1122.A_0025_EPP2316_0003_0018.DIG_Inputs.Input[3] <-> DIG Inputs/Input 4
//     PlcTask Inputs/GVL_iXlinker.EtherCAT_Master_EPPxxxx.Beckhoff_EPP2xxx.Beckhoff_EPP2xxxEK1122.A_0025_EPP2316_0003_0018.DIG_Inputs.Input[4] <-> DIG Inputs/Input 5
//     PlcTask Inputs/GVL_iXlinker.EtherCAT_Master_EPPxxxx.Beckhoff_EPP2xxx.Beckhoff_EPP2xxxEK1122.A_0025_EPP2316_0003_0018.DIG_Inputs.Input[5] <-> DIG Inputs/Input 6
//     PlcTask Inputs/GVL_iXlinker.EtherCAT_Master_EPPxxxx.Beckhoff_EPP2xxx.Beckhoff_EPP2xxxEK1122.A_0025_EPP2316_0003_0018.DIG_Inputs.Input[6] <-> DIG Inputs/Input 7
//     PlcTask Inputs/GVL_iXlinker.EtherCAT_Master_EPPxxxx.Beckhoff_EPP2xxx.Beckhoff_EPP2xxxEK1122.A_0025_EPP2316_0003_0018.DIG_Inputs.Input[7] <-> DIG Inputs/Input 8
//     PlcTask Inputs/GVL_iXlinker.EtherCAT_Master_EPPxxxx.Beckhoff_EPP2xxx.Beckhoff_EPP2xxxEK1122.A_0025_EPP2316_0003_0018.DIG_Inputs.Sync_error <-> DIG Inputs/Sync error
//     PlcTask Inputs/GVL_iXlinker.EtherCAT_Master_EPPxxxx.Beckhoff_EPP2xxx.Beckhoff_EPP2xxxEK1122.A_0025_EPP2316_0003_0018.DIG_Diag_Inputs.Diag_Input[0] <-> DIG Diag Inputs/Diag Input 1
//     PlcTask Inputs/GVL_iXlinker.EtherCAT_Master_EPPxxxx.Beckhoff_EPP2xxx.Beckhoff_EPP2xxxEK1122.A_0025_EPP2316_0003_0018.DIG_Diag_Inputs.Diag_Input[1] <-> DIG Diag Inputs/Diag Input 2
//     PlcTask Inputs/GVL_iXlinker.EtherCAT_Master_EPPxxxx.Beckhoff_EPP2xxx.Beckhoff_EPP2xxxEK1122.A_0025_EPP2316_0003_0018.DIG_Diag_Inputs.Diag_Input[2] <-> DIG Diag Inputs/Diag Input 3
//     PlcTask Inputs/GVL_iXlinker.EtherCAT_Master_EPPxxxx.Beckhoff_EPP2xxx.Beckhoff_EPP2xxxEK1122.A_0025_EPP2316_0003_0018.DIG_Diag_Inputs.Diag_Input[3] <-> DIG Diag Inputs/Diag Input 4
//     PlcTask Inputs/GVL_iXlinker.EtherCAT_Master_EPPxxxx.Beckhoff_EPP2xxx.Beckhoff_EPP2xxxEK1122.A_0025_EPP2316_0003_0018.DIG_Diag_Inputs.Diag_Input[4] <-> DIG Diag Inputs/Diag Input 5
//     PlcTask Inputs/GVL_iXlinker.EtherCAT_Master_EPPxxxx.Beckhoff_EPP2xxx.Beckhoff_EPP2xxxEK1122.A_0025_EPP2316_0003_0018.DIG_Diag_Inputs.Diag_Input[5] <-> DIG Diag Inputs/Diag Input 6
//     PlcTask Inputs/GVL_iXlinker.EtherCAT_Master_EPPxxxx.Beckhoff_EPP2xxx.Beckhoff_EPP2xxxEK1122.A_0025_EPP2316_0003_0018.DIG_Diag_Inputs.Diag_Input[6] <-> DIG Diag Inputs/Diag Input 7
//     PlcTask Inputs/GVL_iXlinker.EtherCAT_Master_EPPxxxx.Beckhoff_EPP2xxx.Beckhoff_EPP2xxxEK1122.A_0025_EPP2316_0003_0018.DIG_Diag_Inputs.Diag_Input[7] <-> DIG Diag Inputs/Diag Input 8
//     PlcTask Inputs/GVL_iXlinker.EtherCAT_Master_EPPxxxx.Beckhoff_EPP2xxx.Beckhoff_EPP2xxxEK1122.A_0025_EPP2316_0003_0018.DIG_Inputs_Device.Safe_state_active <-> DIG Inputs Device/Safe state active
//     PlcTask Inputs/GVL_iXlinker.EtherCAT_Master_EPPxxxx.Beckhoff_EPP2xxx.Beckhoff_EPP2xxxEK1122.A_0025_EPP2316_0003_0018.DIG_Inputs_Device.Error_channel[0] <-> DIG Inputs Device/Error channel 1
//     PlcTask Inputs/GVL_iXlinker.EtherCAT_Master_EPPxxxx.Beckhoff_EPP2xxx.Beckhoff_EPP2xxxEK1122.A_0025_EPP2316_0003_0018.DIG_Inputs_Device.Error_channel[1] <-> DIG Inputs Device/Error channel 2
//     PlcTask Inputs/GVL_iXlinker.EtherCAT_Master_EPPxxxx.Beckhoff_EPP2xxx.Beckhoff_EPP2xxxEK1122.A_0025_EPP2316_0003_0018.DIG_Inputs_Device.Sync_error <-> DIG Inputs Device/Sync error
//     PlcTask Inputs/GVL_iXlinker.EtherCAT_Master_EPPxxxx.Beckhoff_EPP2xxx.Beckhoff_EPP2xxxEK1122.A_0025_EPP2316_0003_0018.DIG_Inputs_Device.TxPDO_Toggle <-> DIG Inputs Device/TxPDO Toggle
//     PlcTask Outputs/GVL_iXlinker.EtherCAT_Master_EPPxxxx.Beckhoff_EPP2xxx.Beckhoff_EPP2xxxEK1122.A_0025_EPP2316_0003_0018.DIG_Outputs.Output[0] <-> DIG Outputs/Output 1
//     PlcTask Outputs/GVL_iXlinker.EtherCAT_Master_EPPxxxx.Beckhoff_EPP2xxx.Beckhoff_EPP2xxxEK1122.A_0025_EPP2316_0003_0018.DIG_Outputs.Output[1] <-> DIG Outputs/Output 2
//     PlcTask Outputs/GVL_iXlinker.EtherCAT_Master_EPPxxxx.Beckhoff_EPP2xxx.Beckhoff_EPP2xxxEK1122.A_0025_EPP2316_0003_0018.DIG_Outputs.Output[2] <-> DIG Outputs/Output 3
//     PlcTask Outputs/GVL_iXlinker.EtherCAT_Master_EPPxxxx.Beckhoff_EPP2xxx.Beckhoff_EPP2xxxEK1122.A_0025_EPP2316_0003_0018.DIG_Outputs.Output[3] <-> DIG Outputs/Output 4
//     PlcTask Outputs/GVL_iXlinker.EtherCAT_Master_EPPxxxx.Beckhoff_EPP2xxx.Beckhoff_EPP2xxxEK1122.A_0025_EPP2316_0003_0018.DIG_Outputs.Output[4] <-> DIG Outputs/Output 5
//     PlcTask Outputs/GVL_iXlinker.EtherCAT_Master_EPPxxxx.Beckhoff_EPP2xxx.Beckhoff_EPP2xxxEK1122.A_0025_EPP2316_0003_0018.DIG_Outputs.Output[5] <-> DIG Outputs/Output 6
//     PlcTask Outputs/GVL_iXlinker.EtherCAT_Master_EPPxxxx.Beckhoff_EPP2xxx.Beckhoff_EPP2xxxEK1122.A_0025_EPP2316_0003_0018.DIG_Outputs.Output[6] <-> DIG Outputs/Output 7
//     PlcTask Outputs/GVL_iXlinker.EtherCAT_Master_EPPxxxx.Beckhoff_EPP2xxx.Beckhoff_EPP2xxxEK1122.A_0025_EPP2316_0003_0018.DIG_Outputs.Output[7] <-> DIG Outputs/Output 8
//     PlcTask Outputs/GVL_iXlinker.EtherCAT_Master_EPPxxxx.Beckhoff_EPP2xxx.Beckhoff_EPP2xxxEK1122.A_0025_EPP2316_0003_0018.DIG_Outputs_Device.Set_safe_state <-> DIG Outputs Device/Set safe state
//     PlcTask Outputs/GVL_iXlinker.EtherCAT_Master_EPPxxxx.Beckhoff_EPP2xxx.Beckhoff_EPP2xxxEK1122.A_0025_EPP2316_0003_0018.DIG_Outputs_Device.Reset_outputs <-> DIG Outputs Device/Reset outputs
//     PlcTask Inputs/GVL_iXlinker.EtherCAT_Master_EPPxxxx.Beckhoff_EPP2xxx.Beckhoff_EPP2xxxEK1122.A_0025_EPP2316_0003_0018.WcState.WcState <-> WcState/WcState
//     PlcTask Inputs/GVL_iXlinker.EtherCAT_Master_EPPxxxx.Beckhoff_EPP2xxx.Beckhoff_EPP2xxxEK1122.A_0025_EPP2316_0003_0018.WcState.InputToggle <-> WcState/InputToggle
//     PlcTask Inputs/GVL_iXlinker.EtherCAT_Master_EPPxxxx.Beckhoff_EPP2xxx.Beckhoff_EPP2xxxEK1122.A_0025_EPP2316_0003_0018.InfoData.AdsAddr <-> InfoData/AdsAddr
//     PlcTask Inputs/GVL_iXlinker.EtherCAT_Master_EPPxxxx.Beckhoff_EPP2xxx.Beckhoff_EPP2xxxEK1122.A_0025_EPP2316_0003_0018.InfoData.State <-> InfoData/State
//   PLC/PLC Instance <-> EtherCAT Master EPPxxxx/Beckhoff EPP2xxx/Beckhoff EPP2xxxEK1122/A_0026(EPP2316-0008-0016)
//     PlcTask Inputs/GVL_iXlinker.EtherCAT_Master_EPPxxxx.Beckhoff_EPP2xxx.Beckhoff_EPP2xxxEK1122.A_0026_EPP2316_0008_0016.DIG_Inputs.Input[0] <-> DIG Inputs/Input 1
//     PlcTask Inputs/GVL_iXlinker.EtherCAT_Master_EPPxxxx.Beckhoff_EPP2xxx.Beckhoff_EPP2xxxEK1122.A_0026_EPP2316_0008_0016.DIG_Inputs.Input[1] <-> DIG Inputs/Input 2
//     PlcTask Inputs/GVL_iXlinker.EtherCAT_Master_EPPxxxx.Beckhoff_EPP2xxx.Beckhoff_EPP2xxxEK1122.A_0026_EPP2316_0008_0016.DIG_Inputs.Input[2] <-> DIG Inputs/Input 3
//     PlcTask Inputs/GVL_iXlinker.EtherCAT_Master_EPPxxxx.Beckhoff_EPP2xxx.Beckhoff_EPP2xxxEK1122.A_0026_EPP2316_0008_0016.DIG_Inputs.Input[3] <-> DIG Inputs/Input 4
//     PlcTask Inputs/GVL_iXlinker.EtherCAT_Master_EPPxxxx.Beckhoff_EPP2xxx.Beckhoff_EPP2xxxEK1122.A_0026_EPP2316_0008_0016.DIG_Inputs.Input[4] <-> DIG Inputs/Input 5
//     PlcTask Inputs/GVL_iXlinker.EtherCAT_Master_EPPxxxx.Beckhoff_EPP2xxx.Beckhoff_EPP2xxxEK1122.A_0026_EPP2316_0008_0016.DIG_Inputs.Input[5] <-> DIG Inputs/Input 6
//     PlcTask Inputs/GVL_iXlinker.EtherCAT_Master_EPPxxxx.Beckhoff_EPP2xxx.Beckhoff_EPP2xxxEK1122.A_0026_EPP2316_0008_0016.DIG_Inputs.Input[6] <-> DIG Inputs/Input 7
//     PlcTask Inputs/GVL_iXlinker.EtherCAT_Master_EPPxxxx.Beckhoff_EPP2xxx.Beckhoff_EPP2xxxEK1122.A_0026_EPP2316_0008_0016.DIG_Inputs.Input[7] <-> DIG Inputs/Input 8
//     PlcTask Inputs/GVL_iXlinker.EtherCAT_Master_EPPxxxx.Beckhoff_EPP2xxx.Beckhoff_EPP2xxxEK1122.A_0026_EPP2316_0008_0016.DIG_Inputs.Sync_Error <-> DIG Inputs/Sync Error
//     PlcTask Inputs/GVL_iXlinker.EtherCAT_Master_EPPxxxx.Beckhoff_EPP2xxx.Beckhoff_EPP2xxxEK1122.A_0026_EPP2316_0008_0016.DIG_Diag_Inputs.Diag_Input[0] <-> DIG Diag Inputs/Diag Input 1
//     PlcTask Inputs/GVL_iXlinker.EtherCAT_Master_EPPxxxx.Beckhoff_EPP2xxx.Beckhoff_EPP2xxxEK1122.A_0026_EPP2316_0008_0016.DIG_Diag_Inputs.Diag_Input[1] <-> DIG Diag Inputs/Diag Input 2
//     PlcTask Inputs/GVL_iXlinker.EtherCAT_Master_EPPxxxx.Beckhoff_EPP2xxx.Beckhoff_EPP2xxxEK1122.A_0026_EPP2316_0008_0016.DIG_Diag_Inputs.Diag_Input[2] <-> DIG Diag Inputs/Diag Input 3
//     PlcTask Inputs/GVL_iXlinker.EtherCAT_Master_EPPxxxx.Beckhoff_EPP2xxx.Beckhoff_EPP2xxxEK1122.A_0026_EPP2316_0008_0016.DIG_Diag_Inputs.Diag_Input[3] <-> DIG Diag Inputs/Diag Input 4
//     PlcTask Inputs/GVL_iXlinker.EtherCAT_Master_EPPxxxx.Beckhoff_EPP2xxx.Beckhoff_EPP2xxxEK1122.A_0026_EPP2316_0008_0016.DIG_Diag_Inputs.Diag_Input[4] <-> DIG Diag Inputs/Diag Input 5
//     PlcTask Inputs/GVL_iXlinker.EtherCAT_Master_EPPxxxx.Beckhoff_EPP2xxx.Beckhoff_EPP2xxxEK1122.A_0026_EPP2316_0008_0016.DIG_Diag_Inputs.Diag_Input[5] <-> DIG Diag Inputs/Diag Input 6
//     PlcTask Inputs/GVL_iXlinker.EtherCAT_Master_EPPxxxx.Beckhoff_EPP2xxx.Beckhoff_EPP2xxxEK1122.A_0026_EPP2316_0008_0016.DIG_Diag_Inputs.Diag_Input[6] <-> DIG Diag Inputs/Diag Input 7
//     PlcTask Inputs/GVL_iXlinker.EtherCAT_Master_EPPxxxx.Beckhoff_EPP2xxx.Beckhoff_EPP2xxxEK1122.A_0026_EPP2316_0008_0016.DIG_Diag_Inputs.Diag_Input[7] <-> DIG Diag Inputs/Diag Input 8
//     PlcTask Inputs/GVL_iXlinker.EtherCAT_Master_EPPxxxx.Beckhoff_EPP2xxx.Beckhoff_EPP2xxxEK1122.A_0026_EPP2316_0008_0016.DIG_Inputs_Device.Safe_state_active <-> DIG Inputs Device/Safe state active
//     PlcTask Inputs/GVL_iXlinker.EtherCAT_Master_EPPxxxx.Beckhoff_EPP2xxx.Beckhoff_EPP2xxxEK1122.A_0026_EPP2316_0008_0016.DIG_Inputs_Device.Error_channel[0] <-> DIG Inputs Device/Error channel 1
//     PlcTask Inputs/GVL_iXlinker.EtherCAT_Master_EPPxxxx.Beckhoff_EPP2xxx.Beckhoff_EPP2xxxEK1122.A_0026_EPP2316_0008_0016.DIG_Inputs_Device.Error_channel[1] <-> DIG Inputs Device/Error channel 2
//     PlcTask Inputs/GVL_iXlinker.EtherCAT_Master_EPPxxxx.Beckhoff_EPP2xxx.Beckhoff_EPP2xxxEK1122.A_0026_EPP2316_0008_0016.DIG_Inputs_Device.Sync_error <-> DIG Inputs Device/Sync error
//     PlcTask Inputs/GVL_iXlinker.EtherCAT_Master_EPPxxxx.Beckhoff_EPP2xxx.Beckhoff_EPP2xxxEK1122.A_0026_EPP2316_0008_0016.DIG_Inputs_Device.TxPDO_Toggle <-> DIG Inputs Device/TxPDO Toggle
//     PlcTask Outputs/GVL_iXlinker.EtherCAT_Master_EPPxxxx.Beckhoff_EPP2xxx.Beckhoff_EPP2xxxEK1122.A_0026_EPP2316_0008_0016.DIG_Outputs.Output[0] <-> DIG Outputs/Output 1
//     PlcTask Outputs/GVL_iXlinker.EtherCAT_Master_EPPxxxx.Beckhoff_EPP2xxx.Beckhoff_EPP2xxxEK1122.A_0026_EPP2316_0008_0016.DIG_Outputs.Output[1] <-> DIG Outputs/Output 2
//     PlcTask Outputs/GVL_iXlinker.EtherCAT_Master_EPPxxxx.Beckhoff_EPP2xxx.Beckhoff_EPP2xxxEK1122.A_0026_EPP2316_0008_0016.DIG_Outputs.Output[2] <-> DIG Outputs/Output 3
//     PlcTask Outputs/GVL_iXlinker.EtherCAT_Master_EPPxxxx.Beckhoff_EPP2xxx.Beckhoff_EPP2xxxEK1122.A_0026_EPP2316_0008_0016.DIG_Outputs.Output[3] <-> DIG Outputs/Output 4
//     PlcTask Outputs/GVL_iXlinker.EtherCAT_Master_EPPxxxx.Beckhoff_EPP2xxx.Beckhoff_EPP2xxxEK1122.A_0026_EPP2316_0008_0016.DIG_Outputs.Output[4] <-> DIG Outputs/Output 5
//     PlcTask Outputs/GVL_iXlinker.EtherCAT_Master_EPPxxxx.Beckhoff_EPP2xxx.Beckhoff_EPP2xxxEK1122.A_0026_EPP2316_0008_0016.DIG_Outputs.Output[5] <-> DIG Outputs/Output 6
//     PlcTask Outputs/GVL_iXlinker.EtherCAT_Master_EPPxxxx.Beckhoff_EPP2xxx.Beckhoff_EPP2xxxEK1122.A_0026_EPP2316_0008_0016.DIG_Outputs.Output[6] <-> DIG Outputs/Output 7
//     PlcTask Outputs/GVL_iXlinker.EtherCAT_Master_EPPxxxx.Beckhoff_EPP2xxx.Beckhoff_EPP2xxxEK1122.A_0026_EPP2316_0008_0016.DIG_Outputs.Output[7] <-> DIG Outputs/Output 8
//     PlcTask Outputs/GVL_iXlinker.EtherCAT_Master_EPPxxxx.Beckhoff_EPP2xxx.Beckhoff_EPP2xxxEK1122.A_0026_EPP2316_0008_0016.DIG_Outputs_Device.Set_safe_state <-> DIG Outputs Device/Set safe state
//     PlcTask Outputs/GVL_iXlinker.EtherCAT_Master_EPPxxxx.Beckhoff_EPP2xxx.Beckhoff_EPP2xxxEK1122.A_0026_EPP2316_0008_0016.DIG_Outputs_Device.Reset_outputs <-> DIG Outputs Device/Reset outputs
//     PlcTask Inputs/GVL_iXlinker.EtherCAT_Master_EPPxxxx.Beckhoff_EPP2xxx.Beckhoff_EPP2xxxEK1122.A_0026_EPP2316_0008_0016.WcState.WcState <-> WcState/WcState
//     PlcTask Inputs/GVL_iXlinker.EtherCAT_Master_EPPxxxx.Beckhoff_EPP2xxx.Beckhoff_EPP2xxxEK1122.A_0026_EPP2316_0008_0016.WcState.InputToggle <-> WcState/InputToggle
//     PlcTask Inputs/GVL_iXlinker.EtherCAT_Master_EPPxxxx.Beckhoff_EPP2xxx.Beckhoff_EPP2xxxEK1122.A_0026_EPP2316_0008_0016.InfoData.AdsAddr <-> InfoData/AdsAddr
//     PlcTask Inputs/GVL_iXlinker.EtherCAT_Master_EPPxxxx.Beckhoff_EPP2xxx.Beckhoff_EPP2xxxEK1122.A_0026_EPP2316_0008_0016.InfoData.State <-> InfoData/State
//   PLC/PLC Instance <-> EtherCAT Master EPPxxxx/Beckhoff EPP2xxx/Beckhoff EPP2xxxEK1122/A_0027(EPP2316-0008-0017)
//     PlcTask Inputs/GVL_iXlinker.EtherCAT_Master_EPPxxxx.Beckhoff_EPP2xxx.Beckhoff_EPP2xxxEK1122.A_0027_EPP2316_0008_0017.DIG_Inputs.Input[0] <-> DIG Inputs/Input 1
//     PlcTask Inputs/GVL_iXlinker.EtherCAT_Master_EPPxxxx.Beckhoff_EPP2xxx.Beckhoff_EPP2xxxEK1122.A_0027_EPP2316_0008_0017.DIG_Inputs.Input[1] <-> DIG Inputs/Input 2
//     PlcTask Inputs/GVL_iXlinker.EtherCAT_Master_EPPxxxx.Beckhoff_EPP2xxx.Beckhoff_EPP2xxxEK1122.A_0027_EPP2316_0008_0017.DIG_Inputs.Input[2] <-> DIG Inputs/Input 3
//     PlcTask Inputs/GVL_iXlinker.EtherCAT_Master_EPPxxxx.Beckhoff_EPP2xxx.Beckhoff_EPP2xxxEK1122.A_0027_EPP2316_0008_0017.DIG_Inputs.Input[3] <-> DIG Inputs/Input 4
//     PlcTask Inputs/GVL_iXlinker.EtherCAT_Master_EPPxxxx.Beckhoff_EPP2xxx.Beckhoff_EPP2xxxEK1122.A_0027_EPP2316_0008_0017.DIG_Inputs.Input[4] <-> DIG Inputs/Input 5
//     PlcTask Inputs/GVL_iXlinker.EtherCAT_Master_EPPxxxx.Beckhoff_EPP2xxx.Beckhoff_EPP2xxxEK1122.A_0027_EPP2316_0008_0017.DIG_Inputs.Input[5] <-> DIG Inputs/Input 6
//     PlcTask Inputs/GVL_iXlinker.EtherCAT_Master_EPPxxxx.Beckhoff_EPP2xxx.Beckhoff_EPP2xxxEK1122.A_0027_EPP2316_0008_0017.DIG_Inputs.Input[6] <-> DIG Inputs/Input 7
//     PlcTask Inputs/GVL_iXlinker.EtherCAT_Master_EPPxxxx.Beckhoff_EPP2xxx.Beckhoff_EPP2xxxEK1122.A_0027_EPP2316_0008_0017.DIG_Inputs.Input[7] <-> DIG Inputs/Input 8
//     PlcTask Inputs/GVL_iXlinker.EtherCAT_Master_EPPxxxx.Beckhoff_EPP2xxx.Beckhoff_EPP2xxxEK1122.A_0027_EPP2316_0008_0017.DIG_Inputs.Sync_Error <-> DIG Inputs/Sync Error
//     PlcTask Inputs/GVL_iXlinker.EtherCAT_Master_EPPxxxx.Beckhoff_EPP2xxx.Beckhoff_EPP2xxxEK1122.A_0027_EPP2316_0008_0017.DIG_Diag_Inputs.Diag_Input[0] <-> DIG Diag Inputs/Diag Input 1
//     PlcTask Inputs/GVL_iXlinker.EtherCAT_Master_EPPxxxx.Beckhoff_EPP2xxx.Beckhoff_EPP2xxxEK1122.A_0027_EPP2316_0008_0017.DIG_Diag_Inputs.Diag_Input[1] <-> DIG Diag Inputs/Diag Input 2
//     PlcTask Inputs/GVL_iXlinker.EtherCAT_Master_EPPxxxx.Beckhoff_EPP2xxx.Beckhoff_EPP2xxxEK1122.A_0027_EPP2316_0008_0017.DIG_Diag_Inputs.Diag_Input[2] <-> DIG Diag Inputs/Diag Input 3
//     PlcTask Inputs/GVL_iXlinker.EtherCAT_Master_EPPxxxx.Beckhoff_EPP2xxx.Beckhoff_EPP2xxxEK1122.A_0027_EPP2316_0008_0017.DIG_Diag_Inputs.Diag_Input[3] <-> DIG Diag Inputs/Diag Input 4
//     PlcTask Inputs/GVL_iXlinker.EtherCAT_Master_EPPxxxx.Beckhoff_EPP2xxx.Beckhoff_EPP2xxxEK1122.A_0027_EPP2316_0008_0017.DIG_Diag_Inputs.Diag_Input[4] <-> DIG Diag Inputs/Diag Input 5
//     PlcTask Inputs/GVL_iXlinker.EtherCAT_Master_EPPxxxx.Beckhoff_EPP2xxx.Beckhoff_EPP2xxxEK1122.A_0027_EPP2316_0008_0017.DIG_Diag_Inputs.Diag_Input[5] <-> DIG Diag Inputs/Diag Input 6
//     PlcTask Inputs/GVL_iXlinker.EtherCAT_Master_EPPxxxx.Beckhoff_EPP2xxx.Beckhoff_EPP2xxxEK1122.A_0027_EPP2316_0008_0017.DIG_Diag_Inputs.Diag_Input[6] <-> DIG Diag Inputs/Diag Input 7
//     PlcTask Inputs/GVL_iXlinker.EtherCAT_Master_EPPxxxx.Beckhoff_EPP2xxx.Beckhoff_EPP2xxxEK1122.A_0027_EPP2316_0008_0017.DIG_Diag_Inputs.Diag_Input[7] <-> DIG Diag Inputs/Diag Input 8
//     PlcTask Inputs/GVL_iXlinker.EtherCAT_Master_EPPxxxx.Beckhoff_EPP2xxx.Beckhoff_EPP2xxxEK1122.A_0027_EPP2316_0008_0017.DIG_Inputs_Device.Safe_state_active <-> DIG Inputs Device/Safe state active
//     PlcTask Inputs/GVL_iXlinker.EtherCAT_Master_EPPxxxx.Beckhoff_EPP2xxx.Beckhoff_EPP2xxxEK1122.A_0027_EPP2316_0008_0017.DIG_Inputs_Device.Error_channel[0] <-> DIG Inputs Device/Error channel 1
//     PlcTask Inputs/GVL_iXlinker.EtherCAT_Master_EPPxxxx.Beckhoff_EPP2xxx.Beckhoff_EPP2xxxEK1122.A_0027_EPP2316_0008_0017.DIG_Inputs_Device.Error_channel[1] <-> DIG Inputs Device/Error channel 2
//     PlcTask Inputs/GVL_iXlinker.EtherCAT_Master_EPPxxxx.Beckhoff_EPP2xxx.Beckhoff_EPP2xxxEK1122.A_0027_EPP2316_0008_0017.DIG_Inputs_Device.Sync_error <-> DIG Inputs Device/Sync error
//     PlcTask Inputs/GVL_iXlinker.EtherCAT_Master_EPPxxxx.Beckhoff_EPP2xxx.Beckhoff_EPP2xxxEK1122.A_0027_EPP2316_0008_0017.DIG_Inputs_Device.TxPDO_Toggle <-> DIG Inputs Device/TxPDO Toggle
//     PlcTask Outputs/GVL_iXlinker.EtherCAT_Master_EPPxxxx.Beckhoff_EPP2xxx.Beckhoff_EPP2xxxEK1122.A_0027_EPP2316_0008_0017.DIG_Outputs.Output[0] <-> DIG Outputs/Output 1
//     PlcTask Outputs/GVL_iXlinker.EtherCAT_Master_EPPxxxx.Beckhoff_EPP2xxx.Beckhoff_EPP2xxxEK1122.A_0027_EPP2316_0008_0017.DIG_Outputs.Output[1] <-> DIG Outputs/Output 2
//     PlcTask Outputs/GVL_iXlinker.EtherCAT_Master_EPPxxxx.Beckhoff_EPP2xxx.Beckhoff_EPP2xxxEK1122.A_0027_EPP2316_0008_0017.DIG_Outputs.Output[2] <-> DIG Outputs/Output 3
//     PlcTask Outputs/GVL_iXlinker.EtherCAT_Master_EPPxxxx.Beckhoff_EPP2xxx.Beckhoff_EPP2xxxEK1122.A_0027_EPP2316_0008_0017.DIG_Outputs.Output[3] <-> DIG Outputs/Output 4
//     PlcTask Outputs/GVL_iXlinker.EtherCAT_Master_EPPxxxx.Beckhoff_EPP2xxx.Beckhoff_EPP2xxxEK1122.A_0027_EPP2316_0008_0017.DIG_Outputs.Output[4] <-> DIG Outputs/Output 5
//     PlcTask Outputs/GVL_iXlinker.EtherCAT_Master_EPPxxxx.Beckhoff_EPP2xxx.Beckhoff_EPP2xxxEK1122.A_0027_EPP2316_0008_0017.DIG_Outputs.Output[5] <-> DIG Outputs/Output 6
//     PlcTask Outputs/GVL_iXlinker.EtherCAT_Master_EPPxxxx.Beckhoff_EPP2xxx.Beckhoff_EPP2xxxEK1122.A_0027_EPP2316_0008_0017.DIG_Outputs.Output[6] <-> DIG Outputs/Output 7
//     PlcTask Outputs/GVL_iXlinker.EtherCAT_Master_EPPxxxx.Beckhoff_EPP2xxx.Beckhoff_EPP2xxxEK1122.A_0027_EPP2316_0008_0017.DIG_Outputs.Output[7] <-> DIG Outputs/Output 8
//     PlcTask Outputs/GVL_iXlinker.EtherCAT_Master_EPPxxxx.Beckhoff_EPP2xxx.Beckhoff_EPP2xxxEK1122.A_0027_EPP2316_0008_0017.DIG_Outputs_Device.Set_safe_state <-> DIG Outputs Device/Set safe state
//     PlcTask Outputs/GVL_iXlinker.EtherCAT_Master_EPPxxxx.Beckhoff_EPP2xxx.Beckhoff_EPP2xxxEK1122.A_0027_EPP2316_0008_0017.DIG_Outputs_Device.Reset_outputs <-> DIG Outputs Device/Reset outputs
//     PlcTask Inputs/GVL_iXlinker.EtherCAT_Master_EPPxxxx.Beckhoff_EPP2xxx.Beckhoff_EPP2xxxEK1122.A_0027_EPP2316_0008_0017.WcState.WcState <-> WcState/WcState
//     PlcTask Inputs/GVL_iXlinker.EtherCAT_Master_EPPxxxx.Beckhoff_EPP2xxx.Beckhoff_EPP2xxxEK1122.A_0027_EPP2316_0008_0017.WcState.InputToggle <-> WcState/InputToggle
//     PlcTask Inputs/GVL_iXlinker.EtherCAT_Master_EPPxxxx.Beckhoff_EPP2xxx.Beckhoff_EPP2xxxEK1122.A_0027_EPP2316_0008_0017.InfoData.AdsAddr <-> InfoData/AdsAddr
//     PlcTask Inputs/GVL_iXlinker.EtherCAT_Master_EPPxxxx.Beckhoff_EPP2xxx.Beckhoff_EPP2xxxEK1122.A_0027_EPP2316_0008_0017.InfoData.State <-> InfoData/State
//   PLC/PLC Instance <-> EtherCAT Master EPPxxxx/Beckhoff EPP2xxx/Beckhoff EPP2xxxEK1122/A_0028(EPP2316-0008-0018)
//     PlcTask Inputs/GVL_iXlinker.EtherCAT_Master_EPPxxxx.Beckhoff_EPP2xxx.Beckhoff_EPP2xxxEK1122.A_0028_EPP2316_0008_0018.DIG_Inputs.Input[0] <-> DIG Inputs/Input 1
//     PlcTask Inputs/GVL_iXlinker.EtherCAT_Master_EPPxxxx.Beckhoff_EPP2xxx.Beckhoff_EPP2xxxEK1122.A_0028_EPP2316_0008_0018.DIG_Inputs.Input[1] <-> DIG Inputs/Input 2
//     PlcTask Inputs/GVL_iXlinker.EtherCAT_Master_EPPxxxx.Beckhoff_EPP2xxx.Beckhoff_EPP2xxxEK1122.A_0028_EPP2316_0008_0018.DIG_Inputs.Input[2] <-> DIG Inputs/Input 3
//     PlcTask Inputs/GVL_iXlinker.EtherCAT_Master_EPPxxxx.Beckhoff_EPP2xxx.Beckhoff_EPP2xxxEK1122.A_0028_EPP2316_0008_0018.DIG_Inputs.Input[3] <-> DIG Inputs/Input 4
//     PlcTask Inputs/GVL_iXlinker.EtherCAT_Master_EPPxxxx.Beckhoff_EPP2xxx.Beckhoff_EPP2xxxEK1122.A_0028_EPP2316_0008_0018.DIG_Inputs.Input[4] <-> DIG Inputs/Input 5
//     PlcTask Inputs/GVL_iXlinker.EtherCAT_Master_EPPxxxx.Beckhoff_EPP2xxx.Beckhoff_EPP2xxxEK1122.A_0028_EPP2316_0008_0018.DIG_Inputs.Input[5] <-> DIG Inputs/Input 6
//     PlcTask Inputs/GVL_iXlinker.EtherCAT_Master_EPPxxxx.Beckhoff_EPP2xxx.Beckhoff_EPP2xxxEK1122.A_0028_EPP2316_0008_0018.DIG_Inputs.Input[6] <-> DIG Inputs/Input 7
//     PlcTask Inputs/GVL_iXlinker.EtherCAT_Master_EPPxxxx.Beckhoff_EPP2xxx.Beckhoff_EPP2xxxEK1122.A_0028_EPP2316_0008_0018.DIG_Inputs.Input[7] <-> DIG Inputs/Input 8
//     PlcTask Inputs/GVL_iXlinker.EtherCAT_Master_EPPxxxx.Beckhoff_EPP2xxx.Beckhoff_EPP2xxxEK1122.A_0028_EPP2316_0008_0018.DIG_Inputs.Sync_error <-> DIG Inputs/Sync error
//     PlcTask Inputs/GVL_iXlinker.EtherCAT_Master_EPPxxxx.Beckhoff_EPP2xxx.Beckhoff_EPP2xxxEK1122.A_0028_EPP2316_0008_0018.DIG_Diag_Inputs.Diag_Input[0] <-> DIG Diag Inputs/Diag Input 1
//     PlcTask Inputs/GVL_iXlinker.EtherCAT_Master_EPPxxxx.Beckhoff_EPP2xxx.Beckhoff_EPP2xxxEK1122.A_0028_EPP2316_0008_0018.DIG_Diag_Inputs.Diag_Input[1] <-> DIG Diag Inputs/Diag Input 2
//     PlcTask Inputs/GVL_iXlinker.EtherCAT_Master_EPPxxxx.Beckhoff_EPP2xxx.Beckhoff_EPP2xxxEK1122.A_0028_EPP2316_0008_0018.DIG_Diag_Inputs.Diag_Input[2] <-> DIG Diag Inputs/Diag Input 3
//     PlcTask Inputs/GVL_iXlinker.EtherCAT_Master_EPPxxxx.Beckhoff_EPP2xxx.Beckhoff_EPP2xxxEK1122.A_0028_EPP2316_0008_0018.DIG_Diag_Inputs.Diag_Input[3] <-> DIG Diag Inputs/Diag Input 4
//     PlcTask Inputs/GVL_iXlinker.EtherCAT_Master_EPPxxxx.Beckhoff_EPP2xxx.Beckhoff_EPP2xxxEK1122.A_0028_EPP2316_0008_0018.DIG_Diag_Inputs.Diag_Input[4] <-> DIG Diag Inputs/Diag Input 5
//     PlcTask Inputs/GVL_iXlinker.EtherCAT_Master_EPPxxxx.Beckhoff_EPP2xxx.Beckhoff_EPP2xxxEK1122.A_0028_EPP2316_0008_0018.DIG_Diag_Inputs.Diag_Input[5] <-> DIG Diag Inputs/Diag Input 6
//     PlcTask Inputs/GVL_iXlinker.EtherCAT_Master_EPPxxxx.Beckhoff_EPP2xxx.Beckhoff_EPP2xxxEK1122.A_0028_EPP2316_0008_0018.DIG_Diag_Inputs.Diag_Input[6] <-> DIG Diag Inputs/Diag Input 7
//     PlcTask Inputs/GVL_iXlinker.EtherCAT_Master_EPPxxxx.Beckhoff_EPP2xxx.Beckhoff_EPP2xxxEK1122.A_0028_EPP2316_0008_0018.DIG_Diag_Inputs.Diag_Input[7] <-> DIG Diag Inputs/Diag Input 8
//     PlcTask Inputs/GVL_iXlinker.EtherCAT_Master_EPPxxxx.Beckhoff_EPP2xxx.Beckhoff_EPP2xxxEK1122.A_0028_EPP2316_0008_0018.DIG_Inputs_Device.Safe_state_active <-> DIG Inputs Device/Safe state active
//     PlcTask Inputs/GVL_iXlinker.EtherCAT_Master_EPPxxxx.Beckhoff_EPP2xxx.Beckhoff_EPP2xxxEK1122.A_0028_EPP2316_0008_0018.DIG_Inputs_Device.Error_channel[0] <-> DIG Inputs Device/Error channel 1
//     PlcTask Inputs/GVL_iXlinker.EtherCAT_Master_EPPxxxx.Beckhoff_EPP2xxx.Beckhoff_EPP2xxxEK1122.A_0028_EPP2316_0008_0018.DIG_Inputs_Device.Error_channel[1] <-> DIG Inputs Device/Error channel 2
//     PlcTask Inputs/GVL_iXlinker.EtherCAT_Master_EPPxxxx.Beckhoff_EPP2xxx.Beckhoff_EPP2xxxEK1122.A_0028_EPP2316_0008_0018.DIG_Inputs_Device.Sync_error <-> DIG Inputs Device/Sync error
//     PlcTask Inputs/GVL_iXlinker.EtherCAT_Master_EPPxxxx.Beckhoff_EPP2xxx.Beckhoff_EPP2xxxEK1122.A_0028_EPP2316_0008_0018.DIG_Inputs_Device.TxPDO_Toggle <-> DIG Inputs Device/TxPDO Toggle
//     PlcTask Outputs/GVL_iXlinker.EtherCAT_Master_EPPxxxx.Beckhoff_EPP2xxx.Beckhoff_EPP2xxxEK1122.A_0028_EPP2316_0008_0018.DIG_Outputs.Output[0] <-> DIG Outputs/Output 1
//     PlcTask Outputs/GVL_iXlinker.EtherCAT_Master_EPPxxxx.Beckhoff_EPP2xxx.Beckhoff_EPP2xxxEK1122.A_0028_EPP2316_0008_0018.DIG_Outputs.Output[1] <-> DIG Outputs/Output 2
//     PlcTask Outputs/GVL_iXlinker.EtherCAT_Master_EPPxxxx.Beckhoff_EPP2xxx.Beckhoff_EPP2xxxEK1122.A_0028_EPP2316_0008_0018.DIG_Outputs.Output[2] <-> DIG Outputs/Output 3
//     PlcTask Outputs/GVL_iXlinker.EtherCAT_Master_EPPxxxx.Beckhoff_EPP2xxx.Beckhoff_EPP2xxxEK1122.A_0028_EPP2316_0008_0018.DIG_Outputs.Output[3] <-> DIG Outputs/Output 4
//     PlcTask Outputs/GVL_iXlinker.EtherCAT_Master_EPPxxxx.Beckhoff_EPP2xxx.Beckhoff_EPP2xxxEK1122.A_0028_EPP2316_0008_0018.DIG_Outputs.Output[4] <-> DIG Outputs/Output 5
//     PlcTask Outputs/GVL_iXlinker.EtherCAT_Master_EPPxxxx.Beckhoff_EPP2xxx.Beckhoff_EPP2xxxEK1122.A_0028_EPP2316_0008_0018.DIG_Outputs.Output[5] <-> DIG Outputs/Output 6
//     PlcTask Outputs/GVL_iXlinker.EtherCAT_Master_EPPxxxx.Beckhoff_EPP2xxx.Beckhoff_EPP2xxxEK1122.A_0028_EPP2316_0008_0018.DIG_Outputs.Output[6] <-> DIG Outputs/Output 7
//     PlcTask Outputs/GVL_iXlinker.EtherCAT_Master_EPPxxxx.Beckhoff_EPP2xxx.Beckhoff_EPP2xxxEK1122.A_0028_EPP2316_0008_0018.DIG_Outputs.Output[7] <-> DIG Outputs/Output 8
//     PlcTask Outputs/GVL_iXlinker.EtherCAT_Master_EPPxxxx.Beckhoff_EPP2xxx.Beckhoff_EPP2xxxEK1122.A_0028_EPP2316_0008_0018.DIG_Outputs_Device.Set_safe_state <-> DIG Outputs Device/Set safe state
//     PlcTask Outputs/GVL_iXlinker.EtherCAT_Master_EPPxxxx.Beckhoff_EPP2xxx.Beckhoff_EPP2xxxEK1122.A_0028_EPP2316_0008_0018.DIG_Outputs_Device.Reset_outputs <-> DIG Outputs Device/Reset outputs
//     PlcTask Inputs/GVL_iXlinker.EtherCAT_Master_EPPxxxx.Beckhoff_EPP2xxx.Beckhoff_EPP2xxxEK1122.A_0028_EPP2316_0008_0018.WcState.WcState <-> WcState/WcState
//     PlcTask Inputs/GVL_iXlinker.EtherCAT_Master_EPPxxxx.Beckhoff_EPP2xxx.Beckhoff_EPP2xxxEK1122.A_0028_EPP2316_0008_0018.WcState.InputToggle <-> WcState/InputToggle
//     PlcTask Inputs/GVL_iXlinker.EtherCAT_Master_EPPxxxx.Beckhoff_EPP2xxx.Beckhoff_EPP2xxxEK1122.A_0028_EPP2316_0008_0018.InfoData.AdsAddr <-> InfoData/AdsAddr
//     PlcTask Inputs/GVL_iXlinker.EtherCAT_Master_EPPxxxx.Beckhoff_EPP2xxx.Beckhoff_EPP2xxxEK1122.A_0028_EPP2316_0008_0018.InfoData.State <-> InfoData/State
//   PLC/PLC Instance <-> EtherCAT Master EPPxxxx/Beckhoff EPP2xxx/Beckhoff EPP2xxxEK1122/A_0029(EPP2318-0001-0016)
//     PlcTask Inputs/GVL_iXlinker.EtherCAT_Master_EPPxxxx.Beckhoff_EPP2xxx.Beckhoff_EPP2xxxEK1122.A_0029_EPP2318_0001_0016.Channel_1.Input <-> Channel 1/Input
//     PlcTask Inputs/GVL_iXlinker.EtherCAT_Master_EPPxxxx.Beckhoff_EPP2xxx.Beckhoff_EPP2xxxEK1122.A_0029_EPP2318_0001_0016.Channel_2.Input <-> Channel 2/Input
//     PlcTask Inputs/GVL_iXlinker.EtherCAT_Master_EPPxxxx.Beckhoff_EPP2xxx.Beckhoff_EPP2xxxEK1122.A_0029_EPP2318_0001_0016.Channel_3.Input <-> Channel 3/Input
//     PlcTask Inputs/GVL_iXlinker.EtherCAT_Master_EPPxxxx.Beckhoff_EPP2xxx.Beckhoff_EPP2xxxEK1122.A_0029_EPP2318_0001_0016.Channel_4.Input <-> Channel 4/Input
//     PlcTask Outputs/GVL_iXlinker.EtherCAT_Master_EPPxxxx.Beckhoff_EPP2xxx.Beckhoff_EPP2xxxEK1122.A_0029_EPP2318_0001_0016.Channel_5.Output <-> Channel 5/Output
//     PlcTask Outputs/GVL_iXlinker.EtherCAT_Master_EPPxxxx.Beckhoff_EPP2xxx.Beckhoff_EPP2xxxEK1122.A_0029_EPP2318_0001_0016.Channel_6.Output <-> Channel 6/Output
//     PlcTask Outputs/GVL_iXlinker.EtherCAT_Master_EPPxxxx.Beckhoff_EPP2xxx.Beckhoff_EPP2xxxEK1122.A_0029_EPP2318_0001_0016.Channel_7.Output <-> Channel 7/Output
//     PlcTask Outputs/GVL_iXlinker.EtherCAT_Master_EPPxxxx.Beckhoff_EPP2xxx.Beckhoff_EPP2xxxEK1122.A_0029_EPP2318_0001_0016.Channel_8.Output <-> Channel 8/Output
//     PlcTask Inputs/GVL_iXlinker.EtherCAT_Master_EPPxxxx.Beckhoff_EPP2xxx.Beckhoff_EPP2xxxEK1122.A_0029_EPP2318_0001_0016.WcState.WcState <-> WcState/WcState
//     PlcTask Inputs/GVL_iXlinker.EtherCAT_Master_EPPxxxx.Beckhoff_EPP2xxx.Beckhoff_EPP2xxxEK1122.A_0029_EPP2318_0001_0016.WcState.InputToggle <-> WcState/InputToggle
//     PlcTask Inputs/GVL_iXlinker.EtherCAT_Master_EPPxxxx.Beckhoff_EPP2xxx.Beckhoff_EPP2xxxEK1122.A_0029_EPP2318_0001_0016.InfoData.State <-> InfoData/State
//   PLC/PLC Instance <-> EtherCAT Master EPPxxxx/Beckhoff EPP2xxx/Beckhoff EPP2xxxEK1122/A_0030(EPP2318-0001-0017)
//     PlcTask Inputs/GVL_iXlinker.EtherCAT_Master_EPPxxxx.Beckhoff_EPP2xxx.Beckhoff_EPP2xxxEK1122.A_0030_EPP2318_0001_0017.Channel_1.Input <-> Channel 1/Input
//     PlcTask Inputs/GVL_iXlinker.EtherCAT_Master_EPPxxxx.Beckhoff_EPP2xxx.Beckhoff_EPP2xxxEK1122.A_0030_EPP2318_0001_0017.Channel_2.Input <-> Channel 2/Input
//     PlcTask Inputs/GVL_iXlinker.EtherCAT_Master_EPPxxxx.Beckhoff_EPP2xxx.Beckhoff_EPP2xxxEK1122.A_0030_EPP2318_0001_0017.Channel_3.Input <-> Channel 3/Input
//     PlcTask Inputs/GVL_iXlinker.EtherCAT_Master_EPPxxxx.Beckhoff_EPP2xxx.Beckhoff_EPP2xxxEK1122.A_0030_EPP2318_0001_0017.Channel_4.Input <-> Channel 4/Input
//     PlcTask Outputs/GVL_iXlinker.EtherCAT_Master_EPPxxxx.Beckhoff_EPP2xxx.Beckhoff_EPP2xxxEK1122.A_0030_EPP2318_0001_0017.Channel_5.Output <-> Channel 5/Output
//     PlcTask Outputs/GVL_iXlinker.EtherCAT_Master_EPPxxxx.Beckhoff_EPP2xxx.Beckhoff_EPP2xxxEK1122.A_0030_EPP2318_0001_0017.Channel_6.Output <-> Channel 6/Output
//     PlcTask Outputs/GVL_iXlinker.EtherCAT_Master_EPPxxxx.Beckhoff_EPP2xxx.Beckhoff_EPP2xxxEK1122.A_0030_EPP2318_0001_0017.Channel_7.Output <-> Channel 7/Output
//     PlcTask Outputs/GVL_iXlinker.EtherCAT_Master_EPPxxxx.Beckhoff_EPP2xxx.Beckhoff_EPP2xxxEK1122.A_0030_EPP2318_0001_0017.Channel_8.Output <-> Channel 8/Output
//     PlcTask Inputs/GVL_iXlinker.EtherCAT_Master_EPPxxxx.Beckhoff_EPP2xxx.Beckhoff_EPP2xxxEK1122.A_0030_EPP2318_0001_0017.WcState.WcState <-> WcState/WcState
//     PlcTask Inputs/GVL_iXlinker.EtherCAT_Master_EPPxxxx.Beckhoff_EPP2xxx.Beckhoff_EPP2xxxEK1122.A_0030_EPP2318_0001_0017.WcState.InputToggle <-> WcState/InputToggle
//     PlcTask Inputs/GVL_iXlinker.EtherCAT_Master_EPPxxxx.Beckhoff_EPP2xxx.Beckhoff_EPP2xxxEK1122.A_0030_EPP2318_0001_0017.InfoData.State <-> InfoData/State
//   PLC/PLC Instance <-> EtherCAT Master EPPxxxx/Beckhoff EPP2xxx/Beckhoff EPP2xxxEK1122/A_0031(EPP2318-0001-0018)
//     PlcTask Inputs/GVL_iXlinker.EtherCAT_Master_EPPxxxx.Beckhoff_EPP2xxx.Beckhoff_EPP2xxxEK1122.A_0031_EPP2318_0001_0018.Channel_1.Input <-> Channel 1/Input
//     PlcTask Inputs/GVL_iXlinker.EtherCAT_Master_EPPxxxx.Beckhoff_EPP2xxx.Beckhoff_EPP2xxxEK1122.A_0031_EPP2318_0001_0018.Channel_2.Input <-> Channel 2/Input
//     PlcTask Inputs/GVL_iXlinker.EtherCAT_Master_EPPxxxx.Beckhoff_EPP2xxx.Beckhoff_EPP2xxxEK1122.A_0031_EPP2318_0001_0018.Channel_3.Input <-> Channel 3/Input
//     PlcTask Inputs/GVL_iXlinker.EtherCAT_Master_EPPxxxx.Beckhoff_EPP2xxx.Beckhoff_EPP2xxxEK1122.A_0031_EPP2318_0001_0018.Channel_4.Input <-> Channel 4/Input
//     PlcTask Outputs/GVL_iXlinker.EtherCAT_Master_EPPxxxx.Beckhoff_EPP2xxx.Beckhoff_EPP2xxxEK1122.A_0031_EPP2318_0001_0018.Channel_5.Output <-> Channel 5/Output
//     PlcTask Outputs/GVL_iXlinker.EtherCAT_Master_EPPxxxx.Beckhoff_EPP2xxx.Beckhoff_EPP2xxxEK1122.A_0031_EPP2318_0001_0018.Channel_6.Output <-> Channel 6/Output
//     PlcTask Outputs/GVL_iXlinker.EtherCAT_Master_EPPxxxx.Beckhoff_EPP2xxx.Beckhoff_EPP2xxxEK1122.A_0031_EPP2318_0001_0018.Channel_7.Output <-> Channel 7/Output
//     PlcTask Outputs/GVL_iXlinker.EtherCAT_Master_EPPxxxx.Beckhoff_EPP2xxx.Beckhoff_EPP2xxxEK1122.A_0031_EPP2318_0001_0018.Channel_8.Output <-> Channel 8/Output
//     PlcTask Inputs/GVL_iXlinker.EtherCAT_Master_EPPxxxx.Beckhoff_EPP2xxx.Beckhoff_EPP2xxxEK1122.A_0031_EPP2318_0001_0018.WcState.WcState <-> WcState/WcState
//     PlcTask Inputs/GVL_iXlinker.EtherCAT_Master_EPPxxxx.Beckhoff_EPP2xxx.Beckhoff_EPP2xxxEK1122.A_0031_EPP2318_0001_0018.WcState.InputToggle <-> WcState/InputToggle
//     PlcTask Inputs/GVL_iXlinker.EtherCAT_Master_EPPxxxx.Beckhoff_EPP2xxx.Beckhoff_EPP2xxxEK1122.A_0031_EPP2318_0001_0018.InfoData.State <-> InfoData/State
//   PLC/PLC Instance <-> EtherCAT Master EPPxxxx/Beckhoff EPP2xxx/Beckhoff EPP2xxxEK1122/A_0032(EPP2318-0002-0016)
//     PlcTask Inputs/GVL_iXlinker.EtherCAT_Master_EPPxxxx.Beckhoff_EPP2xxx.Beckhoff_EPP2xxxEK1122.A_0032_EPP2318_0002_0016.Channel_1.Input <-> Channel 1/Input
//     PlcTask Inputs/GVL_iXlinker.EtherCAT_Master_EPPxxxx.Beckhoff_EPP2xxx.Beckhoff_EPP2xxxEK1122.A_0032_EPP2318_0002_0016.Channel_2.Input <-> Channel 2/Input
//     PlcTask Inputs/GVL_iXlinker.EtherCAT_Master_EPPxxxx.Beckhoff_EPP2xxx.Beckhoff_EPP2xxxEK1122.A_0032_EPP2318_0002_0016.Channel_3.Input <-> Channel 3/Input
//     PlcTask Inputs/GVL_iXlinker.EtherCAT_Master_EPPxxxx.Beckhoff_EPP2xxx.Beckhoff_EPP2xxxEK1122.A_0032_EPP2318_0002_0016.Channel_4.Input <-> Channel 4/Input
//     PlcTask Outputs/GVL_iXlinker.EtherCAT_Master_EPPxxxx.Beckhoff_EPP2xxx.Beckhoff_EPP2xxxEK1122.A_0032_EPP2318_0002_0016.Channel_5.Output <-> Channel 5/Output
//     PlcTask Outputs/GVL_iXlinker.EtherCAT_Master_EPPxxxx.Beckhoff_EPP2xxx.Beckhoff_EPP2xxxEK1122.A_0032_EPP2318_0002_0016.Channel_6.Output <-> Channel 6/Output
//     PlcTask Outputs/GVL_iXlinker.EtherCAT_Master_EPPxxxx.Beckhoff_EPP2xxx.Beckhoff_EPP2xxxEK1122.A_0032_EPP2318_0002_0016.Channel_7.Output <-> Channel 7/Output
//     PlcTask Outputs/GVL_iXlinker.EtherCAT_Master_EPPxxxx.Beckhoff_EPP2xxx.Beckhoff_EPP2xxxEK1122.A_0032_EPP2318_0002_0016.Channel_8.Output <-> Channel 8/Output
//     PlcTask Inputs/GVL_iXlinker.EtherCAT_Master_EPPxxxx.Beckhoff_EPP2xxx.Beckhoff_EPP2xxxEK1122.A_0032_EPP2318_0002_0016.WcState.WcState <-> WcState/WcState
//     PlcTask Inputs/GVL_iXlinker.EtherCAT_Master_EPPxxxx.Beckhoff_EPP2xxx.Beckhoff_EPP2xxxEK1122.A_0032_EPP2318_0002_0016.WcState.InputToggle <-> WcState/InputToggle
//     PlcTask Inputs/GVL_iXlinker.EtherCAT_Master_EPPxxxx.Beckhoff_EPP2xxx.Beckhoff_EPP2xxxEK1122.A_0032_EPP2318_0002_0016.InfoData.State <-> InfoData/State
//   PLC/PLC Instance <-> EtherCAT Master EPPxxxx/Beckhoff EPP2xxx/Beckhoff EPP2xxxEK1122/A_0033(EPP2318-0002-0017)
//     PlcTask Inputs/GVL_iXlinker.EtherCAT_Master_EPPxxxx.Beckhoff_EPP2xxx.Beckhoff_EPP2xxxEK1122.A_0033_EPP2318_0002_0017.Channel_1.Input <-> Channel 1/Input
//     PlcTask Inputs/GVL_iXlinker.EtherCAT_Master_EPPxxxx.Beckhoff_EPP2xxx.Beckhoff_EPP2xxxEK1122.A_0033_EPP2318_0002_0017.Channel_2.Input <-> Channel 2/Input
//     PlcTask Inputs/GVL_iXlinker.EtherCAT_Master_EPPxxxx.Beckhoff_EPP2xxx.Beckhoff_EPP2xxxEK1122.A_0033_EPP2318_0002_0017.Channel_3.Input <-> Channel 3/Input
//     PlcTask Inputs/GVL_iXlinker.EtherCAT_Master_EPPxxxx.Beckhoff_EPP2xxx.Beckhoff_EPP2xxxEK1122.A_0033_EPP2318_0002_0017.Channel_4.Input <-> Channel 4/Input
//     PlcTask Outputs/GVL_iXlinker.EtherCAT_Master_EPPxxxx.Beckhoff_EPP2xxx.Beckhoff_EPP2xxxEK1122.A_0033_EPP2318_0002_0017.Channel_5.Output <-> Channel 5/Output
//     PlcTask Outputs/GVL_iXlinker.EtherCAT_Master_EPPxxxx.Beckhoff_EPP2xxx.Beckhoff_EPP2xxxEK1122.A_0033_EPP2318_0002_0017.Channel_6.Output <-> Channel 6/Output
//     PlcTask Outputs/GVL_iXlinker.EtherCAT_Master_EPPxxxx.Beckhoff_EPP2xxx.Beckhoff_EPP2xxxEK1122.A_0033_EPP2318_0002_0017.Channel_7.Output <-> Channel 7/Output
//     PlcTask Outputs/GVL_iXlinker.EtherCAT_Master_EPPxxxx.Beckhoff_EPP2xxx.Beckhoff_EPP2xxxEK1122.A_0033_EPP2318_0002_0017.Channel_8.Output <-> Channel 8/Output
//     PlcTask Inputs/GVL_iXlinker.EtherCAT_Master_EPPxxxx.Beckhoff_EPP2xxx.Beckhoff_EPP2xxxEK1122.A_0033_EPP2318_0002_0017.WcState.WcState <-> WcState/WcState
//     PlcTask Inputs/GVL_iXlinker.EtherCAT_Master_EPPxxxx.Beckhoff_EPP2xxx.Beckhoff_EPP2xxxEK1122.A_0033_EPP2318_0002_0017.WcState.InputToggle <-> WcState/InputToggle
//     PlcTask Inputs/GVL_iXlinker.EtherCAT_Master_EPPxxxx.Beckhoff_EPP2xxx.Beckhoff_EPP2xxxEK1122.A_0033_EPP2318_0002_0017.InfoData.State <-> InfoData/State
//   PLC/PLC Instance <-> EtherCAT Master EPPxxxx/Beckhoff EPP2xxx/Beckhoff EPP2xxxEK1122/A_0034(EPP2318-0002-0018)
//     PlcTask Inputs/GVL_iXlinker.EtherCAT_Master_EPPxxxx.Beckhoff_EPP2xxx.Beckhoff_EPP2xxxEK1122.A_0034_EPP2318_0002_0018.Channel_1.Input <-> Channel 1/Input
//     PlcTask Inputs/GVL_iXlinker.EtherCAT_Master_EPPxxxx.Beckhoff_EPP2xxx.Beckhoff_EPP2xxxEK1122.A_0034_EPP2318_0002_0018.Channel_2.Input <-> Channel 2/Input
//     PlcTask Inputs/GVL_iXlinker.EtherCAT_Master_EPPxxxx.Beckhoff_EPP2xxx.Beckhoff_EPP2xxxEK1122.A_0034_EPP2318_0002_0018.Channel_3.Input <-> Channel 3/Input
//     PlcTask Inputs/GVL_iXlinker.EtherCAT_Master_EPPxxxx.Beckhoff_EPP2xxx.Beckhoff_EPP2xxxEK1122.A_0034_EPP2318_0002_0018.Channel_4.Input <-> Channel 4/Input
//     PlcTask Outputs/GVL_iXlinker.EtherCAT_Master_EPPxxxx.Beckhoff_EPP2xxx.Beckhoff_EPP2xxxEK1122.A_0034_EPP2318_0002_0018.Channel_5.Output <-> Channel 5/Output
//     PlcTask Outputs/GVL_iXlinker.EtherCAT_Master_EPPxxxx.Beckhoff_EPP2xxx.Beckhoff_EPP2xxxEK1122.A_0034_EPP2318_0002_0018.Channel_6.Output <-> Channel 6/Output
//     PlcTask Outputs/GVL_iXlinker.EtherCAT_Master_EPPxxxx.Beckhoff_EPP2xxx.Beckhoff_EPP2xxxEK1122.A_0034_EPP2318_0002_0018.Channel_7.Output <-> Channel 7/Output
//     PlcTask Outputs/GVL_iXlinker.EtherCAT_Master_EPPxxxx.Beckhoff_EPP2xxx.Beckhoff_EPP2xxxEK1122.A_0034_EPP2318_0002_0018.Channel_8.Output <-> Channel 8/Output
//     PlcTask Inputs/GVL_iXlinker.EtherCAT_Master_EPPxxxx.Beckhoff_EPP2xxx.Beckhoff_EPP2xxxEK1122.A_0034_EPP2318_0002_0018.WcState.WcState <-> WcState/WcState
//     PlcTask Inputs/GVL_iXlinker.EtherCAT_Master_EPPxxxx.Beckhoff_EPP2xxx.Beckhoff_EPP2xxxEK1122.A_0034_EPP2318_0002_0018.WcState.InputToggle <-> WcState/InputToggle
//     PlcTask Inputs/GVL_iXlinker.EtherCAT_Master_EPPxxxx.Beckhoff_EPP2xxx.Beckhoff_EPP2xxxEK1122.A_0034_EPP2318_0002_0018.InfoData.State <-> InfoData/State
//   PLC/PLC Instance <-> EtherCAT Master EPPxxxx/Beckhoff EPP2xxx/Beckhoff EPP2xxxEK1122/A_0035(EPP2328-0001-0016)
//     PlcTask Inputs/GVL_iXlinker.EtherCAT_Master_EPPxxxx.Beckhoff_EPP2xxx.Beckhoff_EPP2xxxEK1122.A_0035_EPP2328_0001_0016.Channel_1.Input <-> Channel 1/Input
//     PlcTask Inputs/GVL_iXlinker.EtherCAT_Master_EPPxxxx.Beckhoff_EPP2xxx.Beckhoff_EPP2xxxEK1122.A_0035_EPP2328_0001_0016.Channel_2.Input <-> Channel 2/Input
//     PlcTask Inputs/GVL_iXlinker.EtherCAT_Master_EPPxxxx.Beckhoff_EPP2xxx.Beckhoff_EPP2xxxEK1122.A_0035_EPP2328_0001_0016.Channel_3.Input <-> Channel 3/Input
//     PlcTask Inputs/GVL_iXlinker.EtherCAT_Master_EPPxxxx.Beckhoff_EPP2xxx.Beckhoff_EPP2xxxEK1122.A_0035_EPP2328_0001_0016.Channel_4.Input <-> Channel 4/Input
//     PlcTask Outputs/GVL_iXlinker.EtherCAT_Master_EPPxxxx.Beckhoff_EPP2xxx.Beckhoff_EPP2xxxEK1122.A_0035_EPP2328_0001_0016.Channel_5.Output <-> Channel 5/Output
//     PlcTask Outputs/GVL_iXlinker.EtherCAT_Master_EPPxxxx.Beckhoff_EPP2xxx.Beckhoff_EPP2xxxEK1122.A_0035_EPP2328_0001_0016.Channel_6.Output <-> Channel 6/Output
//     PlcTask Outputs/GVL_iXlinker.EtherCAT_Master_EPPxxxx.Beckhoff_EPP2xxx.Beckhoff_EPP2xxxEK1122.A_0035_EPP2328_0001_0016.Channel_7.Output <-> Channel 7/Output
//     PlcTask Outputs/GVL_iXlinker.EtherCAT_Master_EPPxxxx.Beckhoff_EPP2xxx.Beckhoff_EPP2xxxEK1122.A_0035_EPP2328_0001_0016.Channel_8.Output <-> Channel 8/Output
//     PlcTask Inputs/GVL_iXlinker.EtherCAT_Master_EPPxxxx.Beckhoff_EPP2xxx.Beckhoff_EPP2xxxEK1122.A_0035_EPP2328_0001_0016.WcState.WcState <-> WcState/WcState
//     PlcTask Inputs/GVL_iXlinker.EtherCAT_Master_EPPxxxx.Beckhoff_EPP2xxx.Beckhoff_EPP2xxxEK1122.A_0035_EPP2328_0001_0016.WcState.InputToggle <-> WcState/InputToggle
//     PlcTask Inputs/GVL_iXlinker.EtherCAT_Master_EPPxxxx.Beckhoff_EPP2xxx.Beckhoff_EPP2xxxEK1122.A_0035_EPP2328_0001_0016.InfoData.State <-> InfoData/State
//   PLC/PLC Instance <-> EtherCAT Master EPPxxxx/Beckhoff EPP2xxx/Beckhoff EPP2xxxEK1122/A_0036(EPP2328-0001-0017)
//     PlcTask Inputs/GVL_iXlinker.EtherCAT_Master_EPPxxxx.Beckhoff_EPP2xxx.Beckhoff_EPP2xxxEK1122.A_0036_EPP2328_0001_0017.Channel_1.Input <-> Channel 1/Input
//     PlcTask Inputs/GVL_iXlinker.EtherCAT_Master_EPPxxxx.Beckhoff_EPP2xxx.Beckhoff_EPP2xxxEK1122.A_0036_EPP2328_0001_0017.Channel_2.Input <-> Channel 2/Input
//     PlcTask Inputs/GVL_iXlinker.EtherCAT_Master_EPPxxxx.Beckhoff_EPP2xxx.Beckhoff_EPP2xxxEK1122.A_0036_EPP2328_0001_0017.Channel_3.Input <-> Channel 3/Input
//     PlcTask Inputs/GVL_iXlinker.EtherCAT_Master_EPPxxxx.Beckhoff_EPP2xxx.Beckhoff_EPP2xxxEK1122.A_0036_EPP2328_0001_0017.Channel_4.Input <-> Channel 4/Input
//     PlcTask Outputs/GVL_iXlinker.EtherCAT_Master_EPPxxxx.Beckhoff_EPP2xxx.Beckhoff_EPP2xxxEK1122.A_0036_EPP2328_0001_0017.Channel_5.Output <-> Channel 5/Output
//     PlcTask Outputs/GVL_iXlinker.EtherCAT_Master_EPPxxxx.Beckhoff_EPP2xxx.Beckhoff_EPP2xxxEK1122.A_0036_EPP2328_0001_0017.Channel_6.Output <-> Channel 6/Output
//     PlcTask Outputs/GVL_iXlinker.EtherCAT_Master_EPPxxxx.Beckhoff_EPP2xxx.Beckhoff_EPP2xxxEK1122.A_0036_EPP2328_0001_0017.Channel_7.Output <-> Channel 7/Output
//     PlcTask Outputs/GVL_iXlinker.EtherCAT_Master_EPPxxxx.Beckhoff_EPP2xxx.Beckhoff_EPP2xxxEK1122.A_0036_EPP2328_0001_0017.Channel_8.Output <-> Channel 8/Output
//     PlcTask Inputs/GVL_iXlinker.EtherCAT_Master_EPPxxxx.Beckhoff_EPP2xxx.Beckhoff_EPP2xxxEK1122.A_0036_EPP2328_0001_0017.WcState.WcState <-> WcState/WcState
//     PlcTask Inputs/GVL_iXlinker.EtherCAT_Master_EPPxxxx.Beckhoff_EPP2xxx.Beckhoff_EPP2xxxEK1122.A_0036_EPP2328_0001_0017.WcState.InputToggle <-> WcState/InputToggle
//     PlcTask Inputs/GVL_iXlinker.EtherCAT_Master_EPPxxxx.Beckhoff_EPP2xxx.Beckhoff_EPP2xxxEK1122.A_0036_EPP2328_0001_0017.InfoData.State <-> InfoData/State
//   PLC/PLC Instance <-> EtherCAT Master EPPxxxx/Beckhoff EPP2xxx/Beckhoff EPP2xxxEK1122/A_0037(EPP2328-0001-0018)
//     PlcTask Inputs/GVL_iXlinker.EtherCAT_Master_EPPxxxx.Beckhoff_EPP2xxx.Beckhoff_EPP2xxxEK1122.A_0037_EPP2328_0001_0018.Channel_1.Input <-> Channel 1/Input
//     PlcTask Inputs/GVL_iXlinker.EtherCAT_Master_EPPxxxx.Beckhoff_EPP2xxx.Beckhoff_EPP2xxxEK1122.A_0037_EPP2328_0001_0018.Channel_2.Input <-> Channel 2/Input
//     PlcTask Inputs/GVL_iXlinker.EtherCAT_Master_EPPxxxx.Beckhoff_EPP2xxx.Beckhoff_EPP2xxxEK1122.A_0037_EPP2328_0001_0018.Channel_3.Input <-> Channel 3/Input
//     PlcTask Inputs/GVL_iXlinker.EtherCAT_Master_EPPxxxx.Beckhoff_EPP2xxx.Beckhoff_EPP2xxxEK1122.A_0037_EPP2328_0001_0018.Channel_4.Input <-> Channel 4/Input
//     PlcTask Outputs/GVL_iXlinker.EtherCAT_Master_EPPxxxx.Beckhoff_EPP2xxx.Beckhoff_EPP2xxxEK1122.A_0037_EPP2328_0001_0018.Channel_5.Output <-> Channel 5/Output
//     PlcTask Outputs/GVL_iXlinker.EtherCAT_Master_EPPxxxx.Beckhoff_EPP2xxx.Beckhoff_EPP2xxxEK1122.A_0037_EPP2328_0001_0018.Channel_6.Output <-> Channel 6/Output
//     PlcTask Outputs/GVL_iXlinker.EtherCAT_Master_EPPxxxx.Beckhoff_EPP2xxx.Beckhoff_EPP2xxxEK1122.A_0037_EPP2328_0001_0018.Channel_7.Output <-> Channel 7/Output
//     PlcTask Outputs/GVL_iXlinker.EtherCAT_Master_EPPxxxx.Beckhoff_EPP2xxx.Beckhoff_EPP2xxxEK1122.A_0037_EPP2328_0001_0018.Channel_8.Output <-> Channel 8/Output
//     PlcTask Inputs/GVL_iXlinker.EtherCAT_Master_EPPxxxx.Beckhoff_EPP2xxx.Beckhoff_EPP2xxxEK1122.A_0037_EPP2328_0001_0018.WcState.WcState <-> WcState/WcState
//     PlcTask Inputs/GVL_iXlinker.EtherCAT_Master_EPPxxxx.Beckhoff_EPP2xxx.Beckhoff_EPP2xxxEK1122.A_0037_EPP2328_0001_0018.WcState.InputToggle <-> WcState/InputToggle
//     PlcTask Inputs/GVL_iXlinker.EtherCAT_Master_EPPxxxx.Beckhoff_EPP2xxx.Beckhoff_EPP2xxxEK1122.A_0037_EPP2328_0001_0018.InfoData.State <-> InfoData/State
//   PLC/PLC Instance <-> EtherCAT Master EPPxxxx/Beckhoff EPP2xxx/Beckhoff EPP2xxxEK1122/A_0038(EPP2328-0002-0016)
//     PlcTask Inputs/GVL_iXlinker.EtherCAT_Master_EPPxxxx.Beckhoff_EPP2xxx.Beckhoff_EPP2xxxEK1122.A_0038_EPP2328_0002_0016.Channel_1.Input <-> Channel 1/Input
//     PlcTask Inputs/GVL_iXlinker.EtherCAT_Master_EPPxxxx.Beckhoff_EPP2xxx.Beckhoff_EPP2xxxEK1122.A_0038_EPP2328_0002_0016.Channel_2.Input <-> Channel 2/Input
//     PlcTask Inputs/GVL_iXlinker.EtherCAT_Master_EPPxxxx.Beckhoff_EPP2xxx.Beckhoff_EPP2xxxEK1122.A_0038_EPP2328_0002_0016.Channel_3.Input <-> Channel 3/Input
//     PlcTask Inputs/GVL_iXlinker.EtherCAT_Master_EPPxxxx.Beckhoff_EPP2xxx.Beckhoff_EPP2xxxEK1122.A_0038_EPP2328_0002_0016.Channel_4.Input <-> Channel 4/Input
//     PlcTask Outputs/GVL_iXlinker.EtherCAT_Master_EPPxxxx.Beckhoff_EPP2xxx.Beckhoff_EPP2xxxEK1122.A_0038_EPP2328_0002_0016.Channel_5.Output <-> Channel 5/Output
//     PlcTask Outputs/GVL_iXlinker.EtherCAT_Master_EPPxxxx.Beckhoff_EPP2xxx.Beckhoff_EPP2xxxEK1122.A_0038_EPP2328_0002_0016.Channel_6.Output <-> Channel 6/Output
//     PlcTask Outputs/GVL_iXlinker.EtherCAT_Master_EPPxxxx.Beckhoff_EPP2xxx.Beckhoff_EPP2xxxEK1122.A_0038_EPP2328_0002_0016.Channel_7.Output <-> Channel 7/Output
//     PlcTask Outputs/GVL_iXlinker.EtherCAT_Master_EPPxxxx.Beckhoff_EPP2xxx.Beckhoff_EPP2xxxEK1122.A_0038_EPP2328_0002_0016.Channel_8.Output <-> Channel 8/Output
//     PlcTask Inputs/GVL_iXlinker.EtherCAT_Master_EPPxxxx.Beckhoff_EPP2xxx.Beckhoff_EPP2xxxEK1122.A_0038_EPP2328_0002_0016.WcState.WcState <-> WcState/WcState
//     PlcTask Inputs/GVL_iXlinker.EtherCAT_Master_EPPxxxx.Beckhoff_EPP2xxx.Beckhoff_EPP2xxxEK1122.A_0038_EPP2328_0002_0016.WcState.InputToggle <-> WcState/InputToggle
//     PlcTask Inputs/GVL_iXlinker.EtherCAT_Master_EPPxxxx.Beckhoff_EPP2xxx.Beckhoff_EPP2xxxEK1122.A_0038_EPP2328_0002_0016.InfoData.State <-> InfoData/State
//   PLC/PLC Instance <-> EtherCAT Master EPPxxxx/Beckhoff EPP2xxx/Beckhoff EPP2xxxEK1122/A_0039(EPP2328-0002-0017)
//     PlcTask Inputs/GVL_iXlinker.EtherCAT_Master_EPPxxxx.Beckhoff_EPP2xxx.Beckhoff_EPP2xxxEK1122.A_0039_EPP2328_0002_0017.Channel_1.Input <-> Channel 1/Input
//     PlcTask Inputs/GVL_iXlinker.EtherCAT_Master_EPPxxxx.Beckhoff_EPP2xxx.Beckhoff_EPP2xxxEK1122.A_0039_EPP2328_0002_0017.Channel_2.Input <-> Channel 2/Input
//     PlcTask Inputs/GVL_iXlinker.EtherCAT_Master_EPPxxxx.Beckhoff_EPP2xxx.Beckhoff_EPP2xxxEK1122.A_0039_EPP2328_0002_0017.Channel_3.Input <-> Channel 3/Input
//     PlcTask Inputs/GVL_iXlinker.EtherCAT_Master_EPPxxxx.Beckhoff_EPP2xxx.Beckhoff_EPP2xxxEK1122.A_0039_EPP2328_0002_0017.Channel_4.Input <-> Channel 4/Input
//     PlcTask Outputs/GVL_iXlinker.EtherCAT_Master_EPPxxxx.Beckhoff_EPP2xxx.Beckhoff_EPP2xxxEK1122.A_0039_EPP2328_0002_0017.Channel_5.Output <-> Channel 5/Output
//     PlcTask Outputs/GVL_iXlinker.EtherCAT_Master_EPPxxxx.Beckhoff_EPP2xxx.Beckhoff_EPP2xxxEK1122.A_0039_EPP2328_0002_0017.Channel_6.Output <-> Channel 6/Output
//     PlcTask Outputs/GVL_iXlinker.EtherCAT_Master_EPPxxxx.Beckhoff_EPP2xxx.Beckhoff_EPP2xxxEK1122.A_0039_EPP2328_0002_0017.Channel_7.Output <-> Channel 7/Output
//     PlcTask Outputs/GVL_iXlinker.EtherCAT_Master_EPPxxxx.Beckhoff_EPP2xxx.Beckhoff_EPP2xxxEK1122.A_0039_EPP2328_0002_0017.Channel_8.Output <-> Channel 8/Output
//     PlcTask Inputs/GVL_iXlinker.EtherCAT_Master_EPPxxxx.Beckhoff_EPP2xxx.Beckhoff_EPP2xxxEK1122.A_0039_EPP2328_0002_0017.WcState.WcState <-> WcState/WcState
//     PlcTask Inputs/GVL_iXlinker.EtherCAT_Master_EPPxxxx.Beckhoff_EPP2xxx.Beckhoff_EPP2xxxEK1122.A_0039_EPP2328_0002_0017.WcState.InputToggle <-> WcState/InputToggle
//     PlcTask Inputs/GVL_iXlinker.EtherCAT_Master_EPPxxxx.Beckhoff_EPP2xxx.Beckhoff_EPP2xxxEK1122.A_0039_EPP2328_0002_0017.InfoData.State <-> InfoData/State
//   PLC/PLC Instance <-> EtherCAT Master EPPxxxx/Beckhoff EPP2xxx/Beckhoff EPP2xxxEK1122/A_0040(EPP2328-0002-0018)
//     PlcTask Inputs/GVL_iXlinker.EtherCAT_Master_EPPxxxx.Beckhoff_EPP2xxx.Beckhoff_EPP2xxxEK1122.A_0040_EPP2328_0002_0018.Channel_1.Input <-> Channel 1/Input
//     PlcTask Inputs/GVL_iXlinker.EtherCAT_Master_EPPxxxx.Beckhoff_EPP2xxx.Beckhoff_EPP2xxxEK1122.A_0040_EPP2328_0002_0018.Channel_2.Input <-> Channel 2/Input
//     PlcTask Inputs/GVL_iXlinker.EtherCAT_Master_EPPxxxx.Beckhoff_EPP2xxx.Beckhoff_EPP2xxxEK1122.A_0040_EPP2328_0002_0018.Channel_3.Input <-> Channel 3/Input
//     PlcTask Inputs/GVL_iXlinker.EtherCAT_Master_EPPxxxx.Beckhoff_EPP2xxx.Beckhoff_EPP2xxxEK1122.A_0040_EPP2328_0002_0018.Channel_4.Input <-> Channel 4/Input
//     PlcTask Outputs/GVL_iXlinker.EtherCAT_Master_EPPxxxx.Beckhoff_EPP2xxx.Beckhoff_EPP2xxxEK1122.A_0040_EPP2328_0002_0018.Channel_5.Output <-> Channel 5/Output
//     PlcTask Outputs/GVL_iXlinker.EtherCAT_Master_EPPxxxx.Beckhoff_EPP2xxx.Beckhoff_EPP2xxxEK1122.A_0040_EPP2328_0002_0018.Channel_6.Output <-> Channel 6/Output
//     PlcTask Outputs/GVL_iXlinker.EtherCAT_Master_EPPxxxx.Beckhoff_EPP2xxx.Beckhoff_EPP2xxxEK1122.A_0040_EPP2328_0002_0018.Channel_7.Output <-> Channel 7/Output
//     PlcTask Outputs/GVL_iXlinker.EtherCAT_Master_EPPxxxx.Beckhoff_EPP2xxx.Beckhoff_EPP2xxxEK1122.A_0040_EPP2328_0002_0018.Channel_8.Output <-> Channel 8/Output
//     PlcTask Inputs/GVL_iXlinker.EtherCAT_Master_EPPxxxx.Beckhoff_EPP2xxx.Beckhoff_EPP2xxxEK1122.A_0040_EPP2328_0002_0018.WcState.WcState <-> WcState/WcState
//     PlcTask Inputs/GVL_iXlinker.EtherCAT_Master_EPPxxxx.Beckhoff_EPP2xxx.Beckhoff_EPP2xxxEK1122.A_0040_EPP2328_0002_0018.WcState.InputToggle <-> WcState/InputToggle
//     PlcTask Inputs/GVL_iXlinker.EtherCAT_Master_EPPxxxx.Beckhoff_EPP2xxx.Beckhoff_EPP2xxxEK1122.A_0040_EPP2328_0002_0018.InfoData.State <-> InfoData/State
//   PLC/PLC Instance <-> EtherCAT Master EPPxxxx/Beckhoff EPP2xxx/Beckhoff EPP2xxxEK1122/A_0041(EPP2334-0061-0016)
//     PlcTask Inputs/GVL_iXlinker.EtherCAT_Master_EPPxxxx.Beckhoff_EPP2xxx.Beckhoff_EPP2xxxEK1122.A_0041_EPP2334_0061_0016.Channel_1.Input <-> Channel 1/Input
//     PlcTask Inputs/GVL_iXlinker.EtherCAT_Master_EPPxxxx.Beckhoff_EPP2xxx.Beckhoff_EPP2xxxEK1122.A_0041_EPP2334_0061_0016.Channel_2.Input <-> Channel 2/Input
//     PlcTask Inputs/GVL_iXlinker.EtherCAT_Master_EPPxxxx.Beckhoff_EPP2xxx.Beckhoff_EPP2xxxEK1122.A_0041_EPP2334_0061_0016.Channel_3.Input <-> Channel 3/Input
//     PlcTask Inputs/GVL_iXlinker.EtherCAT_Master_EPPxxxx.Beckhoff_EPP2xxx.Beckhoff_EPP2xxxEK1122.A_0041_EPP2334_0061_0016.Channel_4.Input <-> Channel 4/Input
//     PlcTask Outputs/GVL_iXlinker.EtherCAT_Master_EPPxxxx.Beckhoff_EPP2xxx.Beckhoff_EPP2xxxEK1122.A_0041_EPP2334_0061_0016.Channel_5.Output <-> Channel 5/Output
//     PlcTask Outputs/GVL_iXlinker.EtherCAT_Master_EPPxxxx.Beckhoff_EPP2xxx.Beckhoff_EPP2xxxEK1122.A_0041_EPP2334_0061_0016.Channel_6.Output <-> Channel 6/Output
//     PlcTask Outputs/GVL_iXlinker.EtherCAT_Master_EPPxxxx.Beckhoff_EPP2xxx.Beckhoff_EPP2xxxEK1122.A_0041_EPP2334_0061_0016.Channel_7.Output <-> Channel 7/Output
//     PlcTask Outputs/GVL_iXlinker.EtherCAT_Master_EPPxxxx.Beckhoff_EPP2xxx.Beckhoff_EPP2xxxEK1122.A_0041_EPP2334_0061_0016.Channel_8.Output <-> Channel 8/Output
//     PlcTask Inputs/GVL_iXlinker.EtherCAT_Master_EPPxxxx.Beckhoff_EPP2xxx.Beckhoff_EPP2xxxEK1122.A_0041_EPP2334_0061_0016.WcState.WcState <-> WcState/WcState
//     PlcTask Inputs/GVL_iXlinker.EtherCAT_Master_EPPxxxx.Beckhoff_EPP2xxx.Beckhoff_EPP2xxxEK1122.A_0041_EPP2334_0061_0016.WcState.InputToggle <-> WcState/InputToggle
//     PlcTask Inputs/GVL_iXlinker.EtherCAT_Master_EPPxxxx.Beckhoff_EPP2xxx.Beckhoff_EPP2xxxEK1122.A_0041_EPP2334_0061_0016.InfoData.State <-> InfoData/State
//   PLC/PLC Instance <-> EtherCAT Master EPPxxxx/Beckhoff EPP2xxx/Beckhoff EPP2xxxEK1122/A_0042(EPP2334-0061-0017)
//     PlcTask Inputs/GVL_iXlinker.EtherCAT_Master_EPPxxxx.Beckhoff_EPP2xxx.Beckhoff_EPP2xxxEK1122.A_0042_EPP2334_0061_0017.Channel_1.Input <-> Channel 1/Input
//     PlcTask Inputs/GVL_iXlinker.EtherCAT_Master_EPPxxxx.Beckhoff_EPP2xxx.Beckhoff_EPP2xxxEK1122.A_0042_EPP2334_0061_0017.Channel_2.Input <-> Channel 2/Input
//     PlcTask Inputs/GVL_iXlinker.EtherCAT_Master_EPPxxxx.Beckhoff_EPP2xxx.Beckhoff_EPP2xxxEK1122.A_0042_EPP2334_0061_0017.Channel_3.Input <-> Channel 3/Input
//     PlcTask Inputs/GVL_iXlinker.EtherCAT_Master_EPPxxxx.Beckhoff_EPP2xxx.Beckhoff_EPP2xxxEK1122.A_0042_EPP2334_0061_0017.Channel_4.Input <-> Channel 4/Input
//     PlcTask Outputs/GVL_iXlinker.EtherCAT_Master_EPPxxxx.Beckhoff_EPP2xxx.Beckhoff_EPP2xxxEK1122.A_0042_EPP2334_0061_0017.Channel_5.Output <-> Channel 5/Output
//     PlcTask Outputs/GVL_iXlinker.EtherCAT_Master_EPPxxxx.Beckhoff_EPP2xxx.Beckhoff_EPP2xxxEK1122.A_0042_EPP2334_0061_0017.Channel_6.Output <-> Channel 6/Output
//     PlcTask Outputs/GVL_iXlinker.EtherCAT_Master_EPPxxxx.Beckhoff_EPP2xxx.Beckhoff_EPP2xxxEK1122.A_0042_EPP2334_0061_0017.Channel_7.Output <-> Channel 7/Output
//     PlcTask Outputs/GVL_iXlinker.EtherCAT_Master_EPPxxxx.Beckhoff_EPP2xxx.Beckhoff_EPP2xxxEK1122.A_0042_EPP2334_0061_0017.Channel_8.Output <-> Channel 8/Output
//     PlcTask Inputs/GVL_iXlinker.EtherCAT_Master_EPPxxxx.Beckhoff_EPP2xxx.Beckhoff_EPP2xxxEK1122.A_0042_EPP2334_0061_0017.WcState.WcState <-> WcState/WcState
//     PlcTask Inputs/GVL_iXlinker.EtherCAT_Master_EPPxxxx.Beckhoff_EPP2xxx.Beckhoff_EPP2xxxEK1122.A_0042_EPP2334_0061_0017.WcState.InputToggle <-> WcState/InputToggle
//     PlcTask Inputs/GVL_iXlinker.EtherCAT_Master_EPPxxxx.Beckhoff_EPP2xxx.Beckhoff_EPP2xxxEK1122.A_0042_EPP2334_0061_0017.InfoData.State <-> InfoData/State
//   PLC/PLC Instance <-> EtherCAT Master EPPxxxx/Beckhoff EPP2xxx/Beckhoff EPP2xxxEK1122/A_0043(EPP2334-0061-0018)
//     PlcTask Inputs/GVL_iXlinker.EtherCAT_Master_EPPxxxx.Beckhoff_EPP2xxx.Beckhoff_EPP2xxxEK1122.A_0043_EPP2334_0061_0018.Channel_1.Input <-> Channel 1/Input
//     PlcTask Inputs/GVL_iXlinker.EtherCAT_Master_EPPxxxx.Beckhoff_EPP2xxx.Beckhoff_EPP2xxxEK1122.A_0043_EPP2334_0061_0018.Channel_2.Input <-> Channel 2/Input
//     PlcTask Inputs/GVL_iXlinker.EtherCAT_Master_EPPxxxx.Beckhoff_EPP2xxx.Beckhoff_EPP2xxxEK1122.A_0043_EPP2334_0061_0018.Channel_3.Input <-> Channel 3/Input
//     PlcTask Inputs/GVL_iXlinker.EtherCAT_Master_EPPxxxx.Beckhoff_EPP2xxx.Beckhoff_EPP2xxxEK1122.A_0043_EPP2334_0061_0018.Channel_4.Input <-> Channel 4/Input
//     PlcTask Outputs/GVL_iXlinker.EtherCAT_Master_EPPxxxx.Beckhoff_EPP2xxx.Beckhoff_EPP2xxxEK1122.A_0043_EPP2334_0061_0018.Channel_5.Output <-> Channel 5/Output
//     PlcTask Outputs/GVL_iXlinker.EtherCAT_Master_EPPxxxx.Beckhoff_EPP2xxx.Beckhoff_EPP2xxxEK1122.A_0043_EPP2334_0061_0018.Channel_6.Output <-> Channel 6/Output
//     PlcTask Outputs/GVL_iXlinker.EtherCAT_Master_EPPxxxx.Beckhoff_EPP2xxx.Beckhoff_EPP2xxxEK1122.A_0043_EPP2334_0061_0018.Channel_7.Output <-> Channel 7/Output
//     PlcTask Outputs/GVL_iXlinker.EtherCAT_Master_EPPxxxx.Beckhoff_EPP2xxx.Beckhoff_EPP2xxxEK1122.A_0043_EPP2334_0061_0018.Channel_8.Output <-> Channel 8/Output
//     PlcTask Inputs/GVL_iXlinker.EtherCAT_Master_EPPxxxx.Beckhoff_EPP2xxx.Beckhoff_EPP2xxxEK1122.A_0043_EPP2334_0061_0018.WcState.WcState <-> WcState/WcState
//     PlcTask Inputs/GVL_iXlinker.EtherCAT_Master_EPPxxxx.Beckhoff_EPP2xxx.Beckhoff_EPP2xxxEK1122.A_0043_EPP2334_0061_0018.WcState.InputToggle <-> WcState/InputToggle
//     PlcTask Inputs/GVL_iXlinker.EtherCAT_Master_EPPxxxx.Beckhoff_EPP2xxx.Beckhoff_EPP2xxxEK1122.A_0043_EPP2334_0061_0018.InfoData.State <-> InfoData/State
//   PLC/PLC Instance <-> EtherCAT Master EPPxxxx/Beckhoff EPP2xxx/Beckhoff EPP2xxxEK1122/A_0044(EPP2334-0061-0019)
//     PlcTask Inputs/GVL_iXlinker.EtherCAT_Master_EPPxxxx.Beckhoff_EPP2xxx.Beckhoff_EPP2xxxEK1122.A_0044_EPP2334_0061_0019.Channel_1.Input <-> Channel 1/Input
//     PlcTask Inputs/GVL_iXlinker.EtherCAT_Master_EPPxxxx.Beckhoff_EPP2xxx.Beckhoff_EPP2xxxEK1122.A_0044_EPP2334_0061_0019.Channel_2.Input <-> Channel 2/Input
//     PlcTask Inputs/GVL_iXlinker.EtherCAT_Master_EPPxxxx.Beckhoff_EPP2xxx.Beckhoff_EPP2xxxEK1122.A_0044_EPP2334_0061_0019.Channel_3.Input <-> Channel 3/Input
//     PlcTask Inputs/GVL_iXlinker.EtherCAT_Master_EPPxxxx.Beckhoff_EPP2xxx.Beckhoff_EPP2xxxEK1122.A_0044_EPP2334_0061_0019.Channel_4.Input <-> Channel 4/Input
//     PlcTask Outputs/GVL_iXlinker.EtherCAT_Master_EPPxxxx.Beckhoff_EPP2xxx.Beckhoff_EPP2xxxEK1122.A_0044_EPP2334_0061_0019.Channel_5.Output <-> Channel 5/Output
//     PlcTask Outputs/GVL_iXlinker.EtherCAT_Master_EPPxxxx.Beckhoff_EPP2xxx.Beckhoff_EPP2xxxEK1122.A_0044_EPP2334_0061_0019.Channel_6.Output <-> Channel 6/Output
//     PlcTask Outputs/GVL_iXlinker.EtherCAT_Master_EPPxxxx.Beckhoff_EPP2xxx.Beckhoff_EPP2xxxEK1122.A_0044_EPP2334_0061_0019.Channel_7.Output <-> Channel 7/Output
//     PlcTask Outputs/GVL_iXlinker.EtherCAT_Master_EPPxxxx.Beckhoff_EPP2xxx.Beckhoff_EPP2xxxEK1122.A_0044_EPP2334_0061_0019.Channel_8.Output <-> Channel 8/Output
//     PlcTask Inputs/GVL_iXlinker.EtherCAT_Master_EPPxxxx.Beckhoff_EPP2xxx.Beckhoff_EPP2xxxEK1122.A_0044_EPP2334_0061_0019.WcState.WcState <-> WcState/WcState
//     PlcTask Inputs/GVL_iXlinker.EtherCAT_Master_EPPxxxx.Beckhoff_EPP2xxx.Beckhoff_EPP2xxxEK1122.A_0044_EPP2334_0061_0019.WcState.InputToggle <-> WcState/InputToggle
//     PlcTask Inputs/GVL_iXlinker.EtherCAT_Master_EPPxxxx.Beckhoff_EPP2xxx.Beckhoff_EPP2xxxEK1122.A_0044_EPP2334_0061_0019.InfoData.State <-> InfoData/State
//   PLC/PLC Instance <-> EtherCAT Master EPPxxxx/Beckhoff EPP2xxx/Beckhoff EPP2xxxEK1122/A_0045(EPP2338-0001-0016)
//     PlcTask Inputs/GVL_iXlinker.EtherCAT_Master_EPPxxxx.Beckhoff_EPP2xxx.Beckhoff_EPP2xxxEK1122.A_0045_EPP2338_0001_0016.Channel_1.Input <-> Channel 1/Input
//     PlcTask Inputs/GVL_iXlinker.EtherCAT_Master_EPPxxxx.Beckhoff_EPP2xxx.Beckhoff_EPP2xxxEK1122.A_0045_EPP2338_0001_0016.Channel_2.Input <-> Channel 2/Input
//     PlcTask Inputs/GVL_iXlinker.EtherCAT_Master_EPPxxxx.Beckhoff_EPP2xxx.Beckhoff_EPP2xxxEK1122.A_0045_EPP2338_0001_0016.Channel_3.Input <-> Channel 3/Input
//     PlcTask Inputs/GVL_iXlinker.EtherCAT_Master_EPPxxxx.Beckhoff_EPP2xxx.Beckhoff_EPP2xxxEK1122.A_0045_EPP2338_0001_0016.Channel_4.Input <-> Channel 4/Input
//     PlcTask Inputs/GVL_iXlinker.EtherCAT_Master_EPPxxxx.Beckhoff_EPP2xxx.Beckhoff_EPP2xxxEK1122.A_0045_EPP2338_0001_0016.Channel_5.Input <-> Channel 5/Input
//     PlcTask Inputs/GVL_iXlinker.EtherCAT_Master_EPPxxxx.Beckhoff_EPP2xxx.Beckhoff_EPP2xxxEK1122.A_0045_EPP2338_0001_0016.Channel_6.Input <-> Channel 6/Input
//     PlcTask Inputs/GVL_iXlinker.EtherCAT_Master_EPPxxxx.Beckhoff_EPP2xxx.Beckhoff_EPP2xxxEK1122.A_0045_EPP2338_0001_0016.Channel_7.Input <-> Channel 7/Input
//     PlcTask Inputs/GVL_iXlinker.EtherCAT_Master_EPPxxxx.Beckhoff_EPP2xxx.Beckhoff_EPP2xxxEK1122.A_0045_EPP2338_0001_0016.Channel_8.Input <-> Channel 8/Input
//     PlcTask Outputs/GVL_iXlinker.EtherCAT_Master_EPPxxxx.Beckhoff_EPP2xxx.Beckhoff_EPP2xxxEK1122.A_0045_EPP2338_0001_0016.Channel_9.Output <-> Channel 9/Output
//     PlcTask Outputs/GVL_iXlinker.EtherCAT_Master_EPPxxxx.Beckhoff_EPP2xxx.Beckhoff_EPP2xxxEK1122.A_0045_EPP2338_0001_0016.Channel_10.Output <-> Channel 10/Output
//     PlcTask Outputs/GVL_iXlinker.EtherCAT_Master_EPPxxxx.Beckhoff_EPP2xxx.Beckhoff_EPP2xxxEK1122.A_0045_EPP2338_0001_0016.Channel_11.Output <-> Channel 11/Output
//     PlcTask Outputs/GVL_iXlinker.EtherCAT_Master_EPPxxxx.Beckhoff_EPP2xxx.Beckhoff_EPP2xxxEK1122.A_0045_EPP2338_0001_0016.Channel_12.Output <-> Channel 12/Output
//     PlcTask Outputs/GVL_iXlinker.EtherCAT_Master_EPPxxxx.Beckhoff_EPP2xxx.Beckhoff_EPP2xxxEK1122.A_0045_EPP2338_0001_0016.Channel_13.Output <-> Channel 13/Output
//     PlcTask Outputs/GVL_iXlinker.EtherCAT_Master_EPPxxxx.Beckhoff_EPP2xxx.Beckhoff_EPP2xxxEK1122.A_0045_EPP2338_0001_0016.Channel_14.Output <-> Channel 14/Output
//     PlcTask Outputs/GVL_iXlinker.EtherCAT_Master_EPPxxxx.Beckhoff_EPP2xxx.Beckhoff_EPP2xxxEK1122.A_0045_EPP2338_0001_0016.Channel_15.Output <-> Channel 15/Output
//     PlcTask Outputs/GVL_iXlinker.EtherCAT_Master_EPPxxxx.Beckhoff_EPP2xxx.Beckhoff_EPP2xxxEK1122.A_0045_EPP2338_0001_0016.Channel_16.Output <-> Channel 16/Output
//     PlcTask Inputs/GVL_iXlinker.EtherCAT_Master_EPPxxxx.Beckhoff_EPP2xxx.Beckhoff_EPP2xxxEK1122.A_0045_EPP2338_0001_0016.WcState.WcState <-> WcState/WcState
//     PlcTask Inputs/GVL_iXlinker.EtherCAT_Master_EPPxxxx.Beckhoff_EPP2xxx.Beckhoff_EPP2xxxEK1122.A_0045_EPP2338_0001_0016.WcState.InputToggle <-> WcState/InputToggle
//     PlcTask Inputs/GVL_iXlinker.EtherCAT_Master_EPPxxxx.Beckhoff_EPP2xxx.Beckhoff_EPP2xxxEK1122.A_0045_EPP2338_0001_0016.InfoData.State <-> InfoData/State
//   PLC/PLC Instance <-> EtherCAT Master EPPxxxx/Beckhoff EPP2xxx/Beckhoff EPP2xxxEK1122/A_0046(EPP2338-0001-0017)
//     PlcTask Inputs/GVL_iXlinker.EtherCAT_Master_EPPxxxx.Beckhoff_EPP2xxx.Beckhoff_EPP2xxxEK1122.A_0046_EPP2338_0001_0017.Channel_1.Input <-> Channel 1/Input
//     PlcTask Inputs/GVL_iXlinker.EtherCAT_Master_EPPxxxx.Beckhoff_EPP2xxx.Beckhoff_EPP2xxxEK1122.A_0046_EPP2338_0001_0017.Channel_2.Input <-> Channel 2/Input
//     PlcTask Inputs/GVL_iXlinker.EtherCAT_Master_EPPxxxx.Beckhoff_EPP2xxx.Beckhoff_EPP2xxxEK1122.A_0046_EPP2338_0001_0017.Channel_3.Input <-> Channel 3/Input
//     PlcTask Inputs/GVL_iXlinker.EtherCAT_Master_EPPxxxx.Beckhoff_EPP2xxx.Beckhoff_EPP2xxxEK1122.A_0046_EPP2338_0001_0017.Channel_4.Input <-> Channel 4/Input
//     PlcTask Inputs/GVL_iXlinker.EtherCAT_Master_EPPxxxx.Beckhoff_EPP2xxx.Beckhoff_EPP2xxxEK1122.A_0046_EPP2338_0001_0017.Channel_5.Input <-> Channel 5/Input
//     PlcTask Inputs/GVL_iXlinker.EtherCAT_Master_EPPxxxx.Beckhoff_EPP2xxx.Beckhoff_EPP2xxxEK1122.A_0046_EPP2338_0001_0017.Channel_6.Input <-> Channel 6/Input
//     PlcTask Inputs/GVL_iXlinker.EtherCAT_Master_EPPxxxx.Beckhoff_EPP2xxx.Beckhoff_EPP2xxxEK1122.A_0046_EPP2338_0001_0017.Channel_7.Input <-> Channel 7/Input
//     PlcTask Inputs/GVL_iXlinker.EtherCAT_Master_EPPxxxx.Beckhoff_EPP2xxx.Beckhoff_EPP2xxxEK1122.A_0046_EPP2338_0001_0017.Channel_8.Input <-> Channel 8/Input
//     PlcTask Outputs/GVL_iXlinker.EtherCAT_Master_EPPxxxx.Beckhoff_EPP2xxx.Beckhoff_EPP2xxxEK1122.A_0046_EPP2338_0001_0017.Channel_9.Output <-> Channel 9/Output
//     PlcTask Outputs/GVL_iXlinker.EtherCAT_Master_EPPxxxx.Beckhoff_EPP2xxx.Beckhoff_EPP2xxxEK1122.A_0046_EPP2338_0001_0017.Channel_10.Output <-> Channel 10/Output
//     PlcTask Outputs/GVL_iXlinker.EtherCAT_Master_EPPxxxx.Beckhoff_EPP2xxx.Beckhoff_EPP2xxxEK1122.A_0046_EPP2338_0001_0017.Channel_11.Output <-> Channel 11/Output
//     PlcTask Outputs/GVL_iXlinker.EtherCAT_Master_EPPxxxx.Beckhoff_EPP2xxx.Beckhoff_EPP2xxxEK1122.A_0046_EPP2338_0001_0017.Channel_12.Output <-> Channel 12/Output
//     PlcTask Outputs/GVL_iXlinker.EtherCAT_Master_EPPxxxx.Beckhoff_EPP2xxx.Beckhoff_EPP2xxxEK1122.A_0046_EPP2338_0001_0017.Channel_13.Output <-> Channel 13/Output
//     PlcTask Outputs/GVL_iXlinker.EtherCAT_Master_EPPxxxx.Beckhoff_EPP2xxx.Beckhoff_EPP2xxxEK1122.A_0046_EPP2338_0001_0017.Channel_14.Output <-> Channel 14/Output
//     PlcTask Outputs/GVL_iXlinker.EtherCAT_Master_EPPxxxx.Beckhoff_EPP2xxx.Beckhoff_EPP2xxxEK1122.A_0046_EPP2338_0001_0017.Channel_15.Output <-> Channel 15/Output
//     PlcTask Outputs/GVL_iXlinker.EtherCAT_Master_EPPxxxx.Beckhoff_EPP2xxx.Beckhoff_EPP2xxxEK1122.A_0046_EPP2338_0001_0017.Channel_16.Output <-> Channel 16/Output
//     PlcTask Inputs/GVL_iXlinker.EtherCAT_Master_EPPxxxx.Beckhoff_EPP2xxx.Beckhoff_EPP2xxxEK1122.A_0046_EPP2338_0001_0017.WcState.WcState <-> WcState/WcState
//     PlcTask Inputs/GVL_iXlinker.EtherCAT_Master_EPPxxxx.Beckhoff_EPP2xxx.Beckhoff_EPP2xxxEK1122.A_0046_EPP2338_0001_0017.WcState.InputToggle <-> WcState/InputToggle
//     PlcTask Inputs/GVL_iXlinker.EtherCAT_Master_EPPxxxx.Beckhoff_EPP2xxx.Beckhoff_EPP2xxxEK1122.A_0046_EPP2338_0001_0017.InfoData.State <-> InfoData/State
//   PLC/PLC Instance <-> EtherCAT Master EPPxxxx/Beckhoff EPP2xxx/Beckhoff EPP2xxxEK1122/A_0047(EPP2338-0001-0018)
//     PlcTask Inputs/GVL_iXlinker.EtherCAT_Master_EPPxxxx.Beckhoff_EPP2xxx.Beckhoff_EPP2xxxEK1122.A_0047_EPP2338_0001_0018.Channel_1.Input <-> Channel 1/Input
//     PlcTask Inputs/GVL_iXlinker.EtherCAT_Master_EPPxxxx.Beckhoff_EPP2xxx.Beckhoff_EPP2xxxEK1122.A_0047_EPP2338_0001_0018.Channel_2.Input <-> Channel 2/Input
//     PlcTask Inputs/GVL_iXlinker.EtherCAT_Master_EPPxxxx.Beckhoff_EPP2xxx.Beckhoff_EPP2xxxEK1122.A_0047_EPP2338_0001_0018.Channel_3.Input <-> Channel 3/Input
//     PlcTask Inputs/GVL_iXlinker.EtherCAT_Master_EPPxxxx.Beckhoff_EPP2xxx.Beckhoff_EPP2xxxEK1122.A_0047_EPP2338_0001_0018.Channel_4.Input <-> Channel 4/Input
//     PlcTask Inputs/GVL_iXlinker.EtherCAT_Master_EPPxxxx.Beckhoff_EPP2xxx.Beckhoff_EPP2xxxEK1122.A_0047_EPP2338_0001_0018.Channel_5.Input <-> Channel 5/Input
//     PlcTask Inputs/GVL_iXlinker.EtherCAT_Master_EPPxxxx.Beckhoff_EPP2xxx.Beckhoff_EPP2xxxEK1122.A_0047_EPP2338_0001_0018.Channel_6.Input <-> Channel 6/Input
//     PlcTask Inputs/GVL_iXlinker.EtherCAT_Master_EPPxxxx.Beckhoff_EPP2xxx.Beckhoff_EPP2xxxEK1122.A_0047_EPP2338_0001_0018.Channel_7.Input <-> Channel 7/Input
//     PlcTask Inputs/GVL_iXlinker.EtherCAT_Master_EPPxxxx.Beckhoff_EPP2xxx.Beckhoff_EPP2xxxEK1122.A_0047_EPP2338_0001_0018.Channel_8.Input <-> Channel 8/Input
//     PlcTask Outputs/GVL_iXlinker.EtherCAT_Master_EPPxxxx.Beckhoff_EPP2xxx.Beckhoff_EPP2xxxEK1122.A_0047_EPP2338_0001_0018.Channel_9.Output <-> Channel 9/Output
//     PlcTask Outputs/GVL_iXlinker.EtherCAT_Master_EPPxxxx.Beckhoff_EPP2xxx.Beckhoff_EPP2xxxEK1122.A_0047_EPP2338_0001_0018.Channel_10.Output <-> Channel 10/Output
//     PlcTask Outputs/GVL_iXlinker.EtherCAT_Master_EPPxxxx.Beckhoff_EPP2xxx.Beckhoff_EPP2xxxEK1122.A_0047_EPP2338_0001_0018.Channel_11.Output <-> Channel 11/Output
//     PlcTask Outputs/GVL_iXlinker.EtherCAT_Master_EPPxxxx.Beckhoff_EPP2xxx.Beckhoff_EPP2xxxEK1122.A_0047_EPP2338_0001_0018.Channel_12.Output <-> Channel 12/Output
//     PlcTask Outputs/GVL_iXlinker.EtherCAT_Master_EPPxxxx.Beckhoff_EPP2xxx.Beckhoff_EPP2xxxEK1122.A_0047_EPP2338_0001_0018.Channel_13.Output <-> Channel 13/Output
//     PlcTask Outputs/GVL_iXlinker.EtherCAT_Master_EPPxxxx.Beckhoff_EPP2xxx.Beckhoff_EPP2xxxEK1122.A_0047_EPP2338_0001_0018.Channel_14.Output <-> Channel 14/Output
//     PlcTask Outputs/GVL_iXlinker.EtherCAT_Master_EPPxxxx.Beckhoff_EPP2xxx.Beckhoff_EPP2xxxEK1122.A_0047_EPP2338_0001_0018.Channel_15.Output <-> Channel 15/Output
//     PlcTask Outputs/GVL_iXlinker.EtherCAT_Master_EPPxxxx.Beckhoff_EPP2xxx.Beckhoff_EPP2xxxEK1122.A_0047_EPP2338_0001_0018.Channel_16.Output <-> Channel 16/Output
//     PlcTask Inputs/GVL_iXlinker.EtherCAT_Master_EPPxxxx.Beckhoff_EPP2xxx.Beckhoff_EPP2xxxEK1122.A_0047_EPP2338_0001_0018.WcState.WcState <-> WcState/WcState
//     PlcTask Inputs/GVL_iXlinker.EtherCAT_Master_EPPxxxx.Beckhoff_EPP2xxx.Beckhoff_EPP2xxxEK1122.A_0047_EPP2338_0001_0018.WcState.InputToggle <-> WcState/InputToggle
//     PlcTask Inputs/GVL_iXlinker.EtherCAT_Master_EPPxxxx.Beckhoff_EPP2xxx.Beckhoff_EPP2xxxEK1122.A_0047_EPP2338_0001_0018.InfoData.State <-> InfoData/State
//   PLC/PLC Instance <-> EtherCAT Master EPPxxxx/Beckhoff EPP2xxx/Beckhoff EPP2xxxEK1122/A_0048(EPP2338-0002-0016)
//     PlcTask Inputs/GVL_iXlinker.EtherCAT_Master_EPPxxxx.Beckhoff_EPP2xxx.Beckhoff_EPP2xxxEK1122.A_0048_EPP2338_0002_0016.Channel_1.Input <-> Channel 1/Input
//     PlcTask Inputs/GVL_iXlinker.EtherCAT_Master_EPPxxxx.Beckhoff_EPP2xxx.Beckhoff_EPP2xxxEK1122.A_0048_EPP2338_0002_0016.Channel_2.Input <-> Channel 2/Input
//     PlcTask Inputs/GVL_iXlinker.EtherCAT_Master_EPPxxxx.Beckhoff_EPP2xxx.Beckhoff_EPP2xxxEK1122.A_0048_EPP2338_0002_0016.Channel_3.Input <-> Channel 3/Input
//     PlcTask Inputs/GVL_iXlinker.EtherCAT_Master_EPPxxxx.Beckhoff_EPP2xxx.Beckhoff_EPP2xxxEK1122.A_0048_EPP2338_0002_0016.Channel_4.Input <-> Channel 4/Input
//     PlcTask Inputs/GVL_iXlinker.EtherCAT_Master_EPPxxxx.Beckhoff_EPP2xxx.Beckhoff_EPP2xxxEK1122.A_0048_EPP2338_0002_0016.Channel_5.Input <-> Channel 5/Input
//     PlcTask Inputs/GVL_iXlinker.EtherCAT_Master_EPPxxxx.Beckhoff_EPP2xxx.Beckhoff_EPP2xxxEK1122.A_0048_EPP2338_0002_0016.Channel_6.Input <-> Channel 6/Input
//     PlcTask Inputs/GVL_iXlinker.EtherCAT_Master_EPPxxxx.Beckhoff_EPP2xxx.Beckhoff_EPP2xxxEK1122.A_0048_EPP2338_0002_0016.Channel_7.Input <-> Channel 7/Input
//     PlcTask Inputs/GVL_iXlinker.EtherCAT_Master_EPPxxxx.Beckhoff_EPP2xxx.Beckhoff_EPP2xxxEK1122.A_0048_EPP2338_0002_0016.Channel_8.Input <-> Channel 8/Input
//     PlcTask Outputs/GVL_iXlinker.EtherCAT_Master_EPPxxxx.Beckhoff_EPP2xxx.Beckhoff_EPP2xxxEK1122.A_0048_EPP2338_0002_0016.Channel_9.Output <-> Channel 9/Output
//     PlcTask Outputs/GVL_iXlinker.EtherCAT_Master_EPPxxxx.Beckhoff_EPP2xxx.Beckhoff_EPP2xxxEK1122.A_0048_EPP2338_0002_0016.Channel_10.Output <-> Channel 10/Output
//     PlcTask Outputs/GVL_iXlinker.EtherCAT_Master_EPPxxxx.Beckhoff_EPP2xxx.Beckhoff_EPP2xxxEK1122.A_0048_EPP2338_0002_0016.Channel_11.Output <-> Channel 11/Output
//     PlcTask Outputs/GVL_iXlinker.EtherCAT_Master_EPPxxxx.Beckhoff_EPP2xxx.Beckhoff_EPP2xxxEK1122.A_0048_EPP2338_0002_0016.Channel_12.Output <-> Channel 12/Output
//     PlcTask Outputs/GVL_iXlinker.EtherCAT_Master_EPPxxxx.Beckhoff_EPP2xxx.Beckhoff_EPP2xxxEK1122.A_0048_EPP2338_0002_0016.Channel_13.Output <-> Channel 13/Output
//     PlcTask Outputs/GVL_iXlinker.EtherCAT_Master_EPPxxxx.Beckhoff_EPP2xxx.Beckhoff_EPP2xxxEK1122.A_0048_EPP2338_0002_0016.Channel_14.Output <-> Channel 14/Output
//     PlcTask Outputs/GVL_iXlinker.EtherCAT_Master_EPPxxxx.Beckhoff_EPP2xxx.Beckhoff_EPP2xxxEK1122.A_0048_EPP2338_0002_0016.Channel_15.Output <-> Channel 15/Output
//     PlcTask Outputs/GVL_iXlinker.EtherCAT_Master_EPPxxxx.Beckhoff_EPP2xxx.Beckhoff_EPP2xxxEK1122.A_0048_EPP2338_0002_0016.Channel_16.Output <-> Channel 16/Output
//     PlcTask Inputs/GVL_iXlinker.EtherCAT_Master_EPPxxxx.Beckhoff_EPP2xxx.Beckhoff_EPP2xxxEK1122.A_0048_EPP2338_0002_0016.WcState.WcState <-> WcState/WcState
//     PlcTask Inputs/GVL_iXlinker.EtherCAT_Master_EPPxxxx.Beckhoff_EPP2xxx.Beckhoff_EPP2xxxEK1122.A_0048_EPP2338_0002_0016.WcState.InputToggle <-> WcState/InputToggle
//     PlcTask Inputs/GVL_iXlinker.EtherCAT_Master_EPPxxxx.Beckhoff_EPP2xxx.Beckhoff_EPP2xxxEK1122.A_0048_EPP2338_0002_0016.InfoData.State <-> InfoData/State
//   PLC/PLC Instance <-> EtherCAT Master EPPxxxx/Beckhoff EPP2xxx/Beckhoff EPP2xxxEK1122/A_0049(EPP2338-0002-0017)
//     PlcTask Inputs/GVL_iXlinker.EtherCAT_Master_EPPxxxx.Beckhoff_EPP2xxx.Beckhoff_EPP2xxxEK1122.A_0049_EPP2338_0002_0017.Channel_1.Input <-> Channel 1/Input
//     PlcTask Inputs/GVL_iXlinker.EtherCAT_Master_EPPxxxx.Beckhoff_EPP2xxx.Beckhoff_EPP2xxxEK1122.A_0049_EPP2338_0002_0017.Channel_2.Input <-> Channel 2/Input
//     PlcTask Inputs/GVL_iXlinker.EtherCAT_Master_EPPxxxx.Beckhoff_EPP2xxx.Beckhoff_EPP2xxxEK1122.A_0049_EPP2338_0002_0017.Channel_3.Input <-> Channel 3/Input
//     PlcTask Inputs/GVL_iXlinker.EtherCAT_Master_EPPxxxx.Beckhoff_EPP2xxx.Beckhoff_EPP2xxxEK1122.A_0049_EPP2338_0002_0017.Channel_4.Input <-> Channel 4/Input
//     PlcTask Inputs/GVL_iXlinker.EtherCAT_Master_EPPxxxx.Beckhoff_EPP2xxx.Beckhoff_EPP2xxxEK1122.A_0049_EPP2338_0002_0017.Channel_5.Input <-> Channel 5/Input
//     PlcTask Inputs/GVL_iXlinker.EtherCAT_Master_EPPxxxx.Beckhoff_EPP2xxx.Beckhoff_EPP2xxxEK1122.A_0049_EPP2338_0002_0017.Channel_6.Input <-> Channel 6/Input
//     PlcTask Inputs/GVL_iXlinker.EtherCAT_Master_EPPxxxx.Beckhoff_EPP2xxx.Beckhoff_EPP2xxxEK1122.A_0049_EPP2338_0002_0017.Channel_7.Input <-> Channel 7/Input
//     PlcTask Inputs/GVL_iXlinker.EtherCAT_Master_EPPxxxx.Beckhoff_EPP2xxx.Beckhoff_EPP2xxxEK1122.A_0049_EPP2338_0002_0017.Channel_8.Input <-> Channel 8/Input
//     PlcTask Outputs/GVL_iXlinker.EtherCAT_Master_EPPxxxx.Beckhoff_EPP2xxx.Beckhoff_EPP2xxxEK1122.A_0049_EPP2338_0002_0017.Channel_9.Output <-> Channel 9/Output
//     PlcTask Outputs/GVL_iXlinker.EtherCAT_Master_EPPxxxx.Beckhoff_EPP2xxx.Beckhoff_EPP2xxxEK1122.A_0049_EPP2338_0002_0017.Channel_10.Output <-> Channel 10/Output
//     PlcTask Outputs/GVL_iXlinker.EtherCAT_Master_EPPxxxx.Beckhoff_EPP2xxx.Beckhoff_EPP2xxxEK1122.A_0049_EPP2338_0002_0017.Channel_11.Output <-> Channel 11/Output
//     PlcTask Outputs/GVL_iXlinker.EtherCAT_Master_EPPxxxx.Beckhoff_EPP2xxx.Beckhoff_EPP2xxxEK1122.A_0049_EPP2338_0002_0017.Channel_12.Output <-> Channel 12/Output
//     PlcTask Outputs/GVL_iXlinker.EtherCAT_Master_EPPxxxx.Beckhoff_EPP2xxx.Beckhoff_EPP2xxxEK1122.A_0049_EPP2338_0002_0017.Channel_13.Output <-> Channel 13/Output
//     PlcTask Outputs/GVL_iXlinker.EtherCAT_Master_EPPxxxx.Beckhoff_EPP2xxx.Beckhoff_EPP2xxxEK1122.A_0049_EPP2338_0002_0017.Channel_14.Output <-> Channel 14/Output
//     PlcTask Outputs/GVL_iXlinker.EtherCAT_Master_EPPxxxx.Beckhoff_EPP2xxx.Beckhoff_EPP2xxxEK1122.A_0049_EPP2338_0002_0017.Channel_15.Output <-> Channel 15/Output
//     PlcTask Outputs/GVL_iXlinker.EtherCAT_Master_EPPxxxx.Beckhoff_EPP2xxx.Beckhoff_EPP2xxxEK1122.A_0049_EPP2338_0002_0017.Channel_16.Output <-> Channel 16/Output
//     PlcTask Inputs/GVL_iXlinker.EtherCAT_Master_EPPxxxx.Beckhoff_EPP2xxx.Beckhoff_EPP2xxxEK1122.A_0049_EPP2338_0002_0017.WcState.WcState <-> WcState/WcState
//     PlcTask Inputs/GVL_iXlinker.EtherCAT_Master_EPPxxxx.Beckhoff_EPP2xxx.Beckhoff_EPP2xxxEK1122.A_0049_EPP2338_0002_0017.WcState.InputToggle <-> WcState/InputToggle
//     PlcTask Inputs/GVL_iXlinker.EtherCAT_Master_EPPxxxx.Beckhoff_EPP2xxx.Beckhoff_EPP2xxxEK1122.A_0049_EPP2338_0002_0017.InfoData.State <-> InfoData/State
//   PLC/PLC Instance <-> EtherCAT Master EPPxxxx/Beckhoff EPP2xxx/Beckhoff EPP2xxxEK1122/A_0050(EPP2338-0002-0018)
//     PlcTask Inputs/GVL_iXlinker.EtherCAT_Master_EPPxxxx.Beckhoff_EPP2xxx.Beckhoff_EPP2xxxEK1122.A_0050_EPP2338_0002_0018.Channel_1.Input <-> Channel 1/Input
//     PlcTask Inputs/GVL_iXlinker.EtherCAT_Master_EPPxxxx.Beckhoff_EPP2xxx.Beckhoff_EPP2xxxEK1122.A_0050_EPP2338_0002_0018.Channel_2.Input <-> Channel 2/Input
//     PlcTask Inputs/GVL_iXlinker.EtherCAT_Master_EPPxxxx.Beckhoff_EPP2xxx.Beckhoff_EPP2xxxEK1122.A_0050_EPP2338_0002_0018.Channel_3.Input <-> Channel 3/Input
//     PlcTask Inputs/GVL_iXlinker.EtherCAT_Master_EPPxxxx.Beckhoff_EPP2xxx.Beckhoff_EPP2xxxEK1122.A_0050_EPP2338_0002_0018.Channel_4.Input <-> Channel 4/Input
//     PlcTask Inputs/GVL_iXlinker.EtherCAT_Master_EPPxxxx.Beckhoff_EPP2xxx.Beckhoff_EPP2xxxEK1122.A_0050_EPP2338_0002_0018.Channel_5.Input <-> Channel 5/Input
//     PlcTask Inputs/GVL_iXlinker.EtherCAT_Master_EPPxxxx.Beckhoff_EPP2xxx.Beckhoff_EPP2xxxEK1122.A_0050_EPP2338_0002_0018.Channel_6.Input <-> Channel 6/Input
//     PlcTask Inputs/GVL_iXlinker.EtherCAT_Master_EPPxxxx.Beckhoff_EPP2xxx.Beckhoff_EPP2xxxEK1122.A_0050_EPP2338_0002_0018.Channel_7.Input <-> Channel 7/Input
//     PlcTask Inputs/GVL_iXlinker.EtherCAT_Master_EPPxxxx.Beckhoff_EPP2xxx.Beckhoff_EPP2xxxEK1122.A_0050_EPP2338_0002_0018.Channel_8.Input <-> Channel 8/Input
//     PlcTask Outputs/GVL_iXlinker.EtherCAT_Master_EPPxxxx.Beckhoff_EPP2xxx.Beckhoff_EPP2xxxEK1122.A_0050_EPP2338_0002_0018.Channel_9.Output <-> Channel 9/Output
//     PlcTask Outputs/GVL_iXlinker.EtherCAT_Master_EPPxxxx.Beckhoff_EPP2xxx.Beckhoff_EPP2xxxEK1122.A_0050_EPP2338_0002_0018.Channel_10.Output <-> Channel 10/Output
//     PlcTask Outputs/GVL_iXlinker.EtherCAT_Master_EPPxxxx.Beckhoff_EPP2xxx.Beckhoff_EPP2xxxEK1122.A_0050_EPP2338_0002_0018.Channel_11.Output <-> Channel 11/Output
//     PlcTask Outputs/GVL_iXlinker.EtherCAT_Master_EPPxxxx.Beckhoff_EPP2xxx.Beckhoff_EPP2xxxEK1122.A_0050_EPP2338_0002_0018.Channel_12.Output <-> Channel 12/Output
//     PlcTask Outputs/GVL_iXlinker.EtherCAT_Master_EPPxxxx.Beckhoff_EPP2xxx.Beckhoff_EPP2xxxEK1122.A_0050_EPP2338_0002_0018.Channel_13.Output <-> Channel 13/Output
